// TIA Portal V19 export
FUNCTION_BLOCK "A0302_Manipolatore_FB"   // FB78, LAD
// stored: MemoryReserve 100, SetENOAutomatically false
   VAR_INPUT
      AreaInterface : "AreaInterface";
      ZSI : "udt_ZoneSafetyInterface";
      DSI_Testa_Feed : "udt_DeviceSafetyInterface";
      DSI_Coda_Feed : "udt_DeviceSafetyInterface";
      DSI_Valve : "udt_DeviceSafetyInterface";
      Drive_Testa : "TAx_DriveInterface";
      Drive_Coda : "TAx_DriveInterface";
      DataIn : Struct
         OP_MoveToPos : Bool;
         Sollevamento : Struct
            OP : "OP_PB";
         END_STRUCT;
         Magneti : Struct
            OP : "OP_PB";
         END_STRUCT;
         Sens : Struct
            Ls1 : Bool;   // Banco di controllo - Ls 1 controllo accumulo pezzi scivolo 1
            Ls2 : Bool;   // Banco di controllo - Ls 2 controllo accumulo pezzi scivolo 2
            Ls3 : Bool;   // Banco di controllo - Ls 3 controllo accumulo pezzi scivolo 3
            Ls4 : Bool;   // Banco di controllo - Ls 4 controllo accumulo pezzi scivolo 4
         END_STRUCT;
      END_STRUCT;
      CIn : Struct
         Manager : Struct
            EnableStopDoorOpeningReq { ExternalAccessible := 'False'; ExternalVisible := 'False'; ExternalWritable := 'False'} : Bool;
            EnableStopInPhase { ExternalAccessible := 'False'; ExternalVisible := 'False'; ExternalWritable := 'False'} : Bool;
            EnableStopProgrammed { ExternalAccessible := 'False'; ExternalVisible := 'False'; ExternalWritable := 'False'} : Bool;
            Control_ON { ExternalAccessible := 'False'; ExternalVisible := 'False'; ExternalWritable := 'False'} : Bool;
            MoveToPos { ExternalAccessible := 'False'; ExternalVisible := 'False'; ExternalWritable := 'False'} : Bool;
            Pos { ExternalAccessible := 'False'; ExternalVisible := 'False'; ExternalWritable := 'False'} : LReal;
            Vel : LReal;
            Acc : LReal;
            Dec : LReal;
            Sollevamento { ExternalAccessible := 'False'; ExternalVisible := 'False'; ExternalWritable := 'False'} : Struct
               Rest : Bool;
               Work : Bool;
            END_STRUCT;
            Magneti { ExternalAccessible := 'False'; ExternalVisible := 'False'; ExternalWritable := 'False'} : Struct
               Rest : Bool;
               Work : Bool;
            END_STRUCT;
         END_STRUCT;
         OP_SemiAut_PB { ExternalWritable := 'False'} : Bool;
         Rulliera { ExternalWritable := 'False'} : Struct
            Centratori : "ValveMachine_COut";
            Coda : Struct
               Sens : Struct
                  FTC_Rall : Bool;   // Sensori presenza materiale banco rallentamento ingresso
                  FTC_Prox_Ing : Bool;   // Sensori presenza materiale banco limite ingresso
               END_STRUCT;
            END_STRUCT;
            Centro : Struct
               Sens : Struct
                  FTC_Centrale : Bool;   // 2010BF1 - I50.2
               END_STRUCT;
            END_STRUCT;
         END_STRUCT;
         CarroPareggTesta { ExternalWritable := 'False'} : Struct
            Sens : Struct
               FTC1_Rall : Bool;   // 2010BF2 - I50.3
               FTC2_Prox_Ls : Bool;   // 2010BF3 - I50.4
               PresenzaMat : Bool;   // FC presenza materiale agganciato lato paregg testa
            END_STRUCT;
         END_STRUCT;
         CarroPareggCoda { ExternalWritable := 'False'} : Struct
            Sens : Struct
               FTC_Ingombro_In : Bool;   // 2012BF1 - I50.0
               FTC_Ingombro_Out : Bool;   // 2012BF2 - I50.1
               PresenzaMat : Bool;   // FC presenza materiale agganciato lato paregg coda
            END_STRUCT;
         END_STRUCT;
         CarriPareggiatori : Struct
            ZoneA0302Entry_Empty { ExternalWritable := 'False'} : Bool;
            ZoneA0302Exit_Empty { ExternalWritable := 'False'} : Bool;
            RequestNewPosition : Bool;
         END_STRUCT;
         Spalle : Struct
            Coda : Struct
               ActualPos : LReal;
            END_STRUCT;
            Testa : Struct
               ActualPos : LReal;
            END_STRUCT;
         END_STRUCT;
      END_STRUCT;
      Config : Struct
         Testa : Struct
            Ax : "Positioning_EPOS_Machine_Config_NEW";
            Sollevatore : "ValveMachine_Config";
            Magnete : "ValveMachine_Config";
         END_STRUCT;
         Coda : Struct
            Ax : "Positioning_EPOS_Machine_Config_NEW";
            Sollevatore : "ValveMachine_Config";
            Magnete : "ValveMachine_Config";
         END_STRUCT;
         DelayMissingCondition : Time;
      END_STRUCT;
      HWID_AxTesta_TEL111 : HW_SUBMODULE;
      HWID_AxCoda_TEL111 : HW_SUBMODULE;
   END_VAR
   VAR_OUTPUT
      MachineInterface : "MachineInterface";
      COut : Struct
         Testa : Struct
            Ax : "Positioning_EPOS_Machine_COut";
            Sollevatore : "ValveMachine_COut";
            Magnete : "ValveMachine_COut";
         END_STRUCT;
         Coda : Struct
            Ax : "Positioning_EPOS_Machine_COut";
            Sollevatore : "ValveMachine_COut";
            Magnete : "ValveMachine_COut";
         END_STRUCT;
         CheckAxTesta : Struct
            InPos_Prelievo : Bool;
            InPos_BancoScarto : Bool;
            InPos_BancoA0303 : Bool;
         END_STRUCT;
         CheckAxCoda : Struct
            InPos_Prelievo : Bool;
            InPos_BancoScarto : Bool;
            InPos_BancoA0303 : Bool;
         END_STRUCT;
         InPos_Prelievo : Bool;
         InPos_BancoScarto : Bool;
         InPos_BancoA0303 : Bool;
         OutWorkSpace : Bool;   // Fuori ingombro banco A0303
      END_STRUCT;
   END_VAR
   VAR_IN_OUT
      Par : Struct
         Ax : "Positioning_EPOS_Machine_Par";
         Ax_Aut : "A0301_Mach_Speed_Par";
         Ax_Pos : Struct
            Prelievo : LReal;
            BancoCtrl : LReal;
            BancoA0303 : LReal;
            Tollerance : Struct
               Prelievo : LReal;
               BancoCtrl : LReal;
               BancoA0303 : LReal;
            END_STRUCT;
         END_STRUCT;
      END_STRUCT;
      Pers_Data : Struct
         EncoderAbsolute_Preset_OK : Bool;
         Persistent_ActualPosition : LReal;
      END_STRUCT;
   END_VAR
   VAR
      Alarm : Struct
         Testa : Struct
            Ax : "Positioning_EPOS_Machine_Alr";
            Sollevatore : "ValveAlr";
            Magnete : "ValveAlr";
         END_STRUCT;
         Coda : Struct
            Ax : "Positioning_EPOS_Machine_Alr";
            Sollevatore : "ValveAlr";
            Magnete : "ValveAlr";
         END_STRUCT;
         CheckBothAxMove : Bool;
      END_STRUCT;
      Warning : Struct
         Testa : Struct
            Ax : "Positioning_EPOS_Machine_Wng";
            Sollevatore : "ValveMachine_Wng";
            Magnete : "ValveMachine_Wng";
         END_STRUCT;
         Coda : Struct
            Ax : "Positioning_EPOS_Machine_Wng";
            Sollevatore : "ValveMachine_Wng";
            Magnete : "ValveMachine_Wng";
         END_STRUCT;
         MissingCnd : Struct
            OP_REST_Sollevamento : Bool;   // Mancanza comando arresto
            OP_WORK_Sollevamento : Bool;   // Mancanza consenso lavoro
            OP_REST_Magneti : Bool;   // Mancanza comando arresto
            OP_WORK_Magneti : Bool;   // Mancanza consenso lavoro
         END_STRUCT;
      END_STRUCT;
      HMI : Struct
         Selection : Struct   // 0=Disable / 1=Enable Pin
            Ax : Int;   // 0:Entrambe / 1:Testa / 2:Coda
         END_STRUCT;
         Ax_Testa : "AnalogSens_HmiData";
         Ax_Coda : "AnalogSens_HmiData";
      END_STRUCT;
      Sts : Struct
         ReadyForMove : Bool;   // Pronto al movimento
         OP_Manip_CanMoveFreely : Bool;
         OP_Ax_CanMoveFreely : Bool;
         Op_MoveToPos_Cnd : Bool;
         Sollevamento : Struct
            OP_Rest_Cnd : Bool;
            Op_Work_Cnd : Bool;
         END_STRUCT;
         Magneti : Struct
            OP_Rest_Cnd : Bool;
            Op_Work_Cnd : Bool;
         END_STRUCT;
         Coda_PermessoDaSynchOk : Bool;
         Testa_PermessoDaSynchOk : Bool;
      END_STRUCT;
      Ctrl : Struct
         Sollevamento : Struct
            OP_Rest_Man : Bool;
            OP_Work_Man : Bool;
            OP_Rest_Aut : Bool;
            OP_Work_Aut : Bool;
            OP_Rest : Bool;
            OP_Work : Bool;
         END_STRUCT;
         Magneti : Struct
            OP_Rest_Aut : Bool;
            OP_Work_Aut : Bool;
            OP_Rest_Man : Bool;
            OP_Work_Man : Bool;
            OP_Rest : Bool;
            OP_Work : Bool;
         END_STRUCT;
         Ax : Struct
            OP_MoveToPos_Man : Bool;
            OP_MoveToPos_Aut : Bool;
            OP_MoveToPos : Bool;
         END_STRUCT;
      END_STRUCT;
      AUX : Struct
         OP_MoveToPos : Bool;
         Sollevamento : Struct
            OP_Rest : Bool;
            OP_Work : Bool;
         END_STRUCT;
         Magneti : Struct
            OP_Rest : Bool;
            OP_Work : Bool;
         END_STRUCT;
      END_STRUCT;
      Ax_Testa : "Positioning_EPOS_Machine_FB_NEW";
      Ax_Coda : "Positioning_EPOS_Machine_FB_NEW";
      Sollevatore_Testa { S7_SetPoint := 'True'} : "ValveMachine_FB";
      Sollevatore_Coda { S7_SetPoint := 'True'} : "ValveMachine_FB";
      Magnete_Testa { S7_SetPoint := 'True'} : "ValveMachine_FB";
      Magnete_Coda { S7_SetPoint := 'True'} : "ValveMachine_FB";
      TON_Magneti : Struct
         OP_REST_MissingCnd { S7_SetPoint := 'True'} : TON_TIME;
         OP_WORK_MissingCnd { S7_SetPoint := 'True'} : TON_TIME;
      END_STRUCT;
      TON_Sollevamento : Struct
         OP_REST_MissingCnd { S7_SetPoint := 'True'} : TON_TIME;
         OP_WORK_MissingCnd { S7_SetPoint := 'True'} : TON_TIME;
      END_STRUCT;
      TON_CheckAxMove : IEC_TIMER;
      CheckAxisSynch { ExternalAccessible := 'False'; ExternalVisible := 'False'; ExternalWritable := 'False'} : "CheckAxisSynch";
      Sts_PosAxis { S7_SetPoint := 'True'} : Int;
   END_VAR
   VAR_TEMP
      PE : Struct
         OP_MoveToPos : Bool;
         Sollevamento : Struct
            OP_Rest : Bool;
            OP_Work : Bool;
         END_STRUCT;
         Magneti : Struct
            OP_Rest : Bool;
            OP_Work : Bool;
         END_STRUCT;
      END_STRUCT;
   END_VAR
   VAR CONSTANT
      MaxDistance : LReal := 5.0;
      MinDistance : LReal := 0.7;   // soglia inferiore per isteresi
   END_VAR
   VAR_TEMP   // added for the SCL form of the ladder/FBD networks
      _w1 : Bool;
      _w2 : Bool;
      _w3 : Bool;
      _w4 : Bool;
      _w5 : Bool;
      _w6 : Bool;
      _w7 : Bool;
      _w8 : Bool;
      _w9 : Bool;
   END_VAR
BEGIN

REGION Network 1 (SCL): Reset allarmi
   IF #AreaInterface.RstAlarms THEN
       #Alarm.CheckBothAxMove:=FALSE;
       #Warning.Testa.Ax.Minus_CndMissing := FALSE;
       #Warning.Testa.Ax.Plus_CndMissing := FALSE;
       #Warning.Coda.Ax.Minus_CndMissing := FALSE;
       #Warning.Coda.Ax.Plus_CndMissing := FALSE;
   END_IF;
END_REGION

REGION Network 3 (SCL): PrjConfig - GESTIONE PARAMETRI MANIPOLATORI
   // Asse MANIPOLATORI









   // SOLLEVATORE
   // 







   // MAGNETE
   //
END_REGION

REGION Network 5: [Ax] - Controllo posizione dei Manipolatori In PRELIEVO su PAREGGIATORI
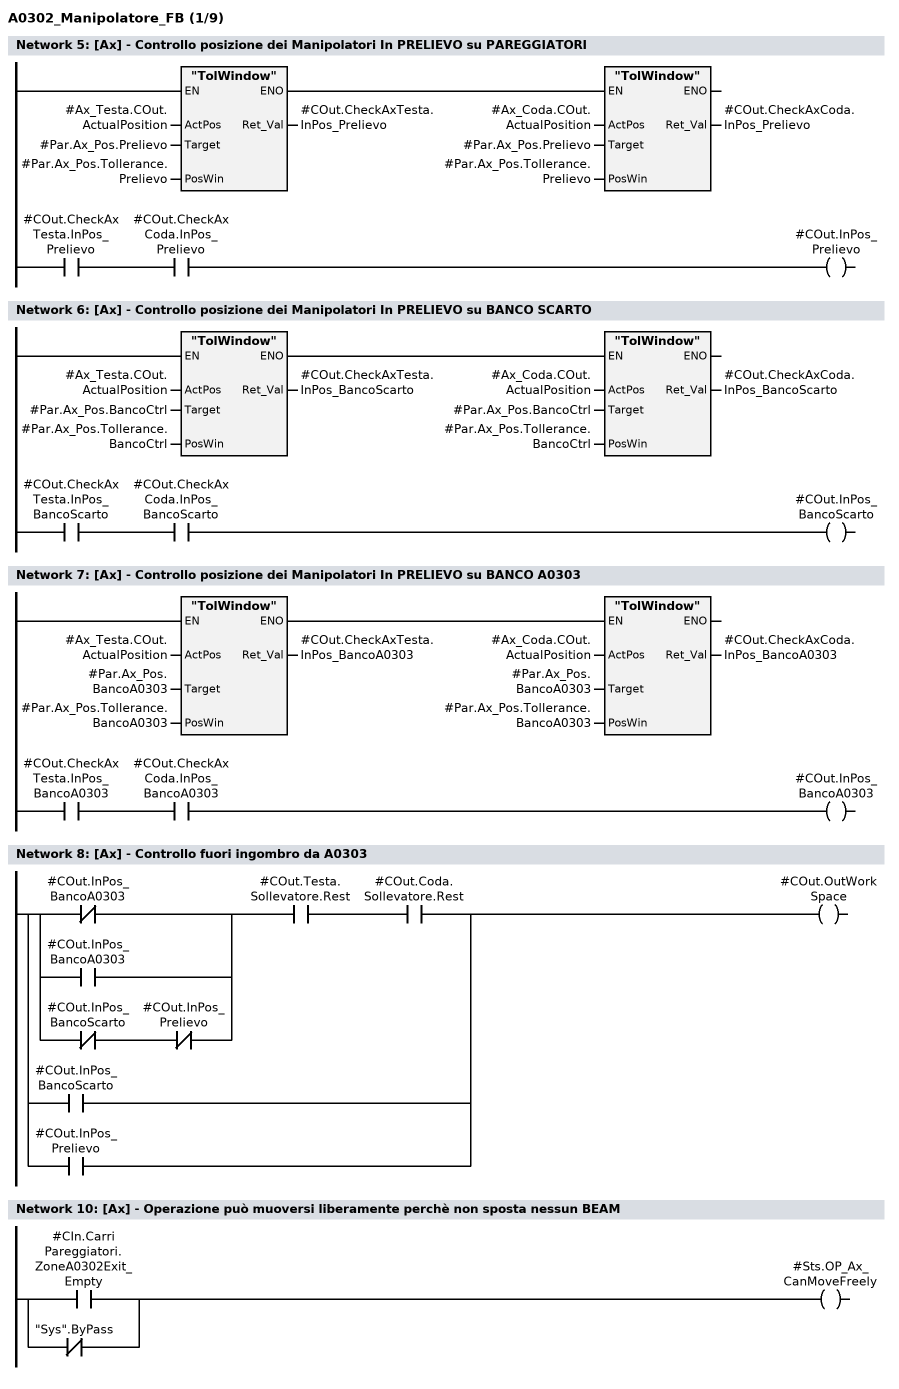
   RUNG wire#powerrail
      "TolWindow"(ActPos := #Ax_Testa.COut.ActualPosition, Target := #Par.Ax_Pos.Prelievo, PosWin := #Par.Ax_Pos.Tollerance.Prelievo, Ret_Val => #COut.CheckAxTesta.InPos_Prelievo)
      "TolWindow"(ActPos := #Ax_Coda.COut.ActualPosition, Target := #Par.Ax_Pos.Prelievo, PosWin := #Par.Ax_Pos.Tollerance.Prelievo, Ret_Val => #COut.CheckAxCoda.InPos_Prelievo)
   END_RUNG
   RUNG wire#powerrail
      Contact( #COut.CheckAxTesta.InPos_Prelievo )
      Contact( #COut.CheckAxCoda.InPos_Prelievo )
      Coil( #COut.InPos_Prelievo )
   END_RUNG
   // the same network as SCL:
   #COut.CheckAxTesta.InPos_Prelievo := "TolWindow"(ActPos := #Ax_Testa.COut.ActualPosition,
                           Target := #Par.Ax_Pos.Prelievo,
                           PosWin := #Par.Ax_Pos.Tollerance.Prelievo,
                           ENO => #_w1);
   IF #_w1 THEN
       #COut.CheckAxCoda.InPos_Prelievo := "TolWindow"(ActPos := #Ax_Coda.COut.ActualPosition,
                               Target := #Par.Ax_Pos.Prelievo,
                               PosWin := #Par.Ax_Pos.Tollerance.Prelievo);
   END_IF;
   #COut.InPos_Prelievo := #COut.CheckAxTesta.InPos_Prelievo AND #COut.CheckAxCoda.InPos_Prelievo;
END_REGION

REGION Network 6: [Ax] - Controllo posizione dei Manipolatori In PRELIEVO su BANCO SCARTO
   RUNG wire#powerrail
      "TolWindow"(ActPos := #Ax_Testa.COut.ActualPosition, Target := #Par.Ax_Pos.BancoCtrl, PosWin := #Par.Ax_Pos.Tollerance.BancoCtrl, Ret_Val => #COut.CheckAxTesta.InPos_BancoScarto)
      "TolWindow"(ActPos := #Ax_Coda.COut.ActualPosition, Target := #Par.Ax_Pos.BancoCtrl, PosWin := #Par.Ax_Pos.Tollerance.BancoCtrl, Ret_Val => #COut.CheckAxCoda.InPos_BancoScarto)
   END_RUNG
   RUNG wire#powerrail
      Contact( #COut.CheckAxTesta.InPos_BancoScarto )
      Contact( #COut.CheckAxCoda.InPos_BancoScarto )
      Coil( #COut.InPos_BancoScarto )
   END_RUNG
   // the same network as SCL:
   #COut.CheckAxTesta.InPos_BancoScarto := "TolWindow"(ActPos := #Ax_Testa.COut.ActualPosition,
                           Target := #Par.Ax_Pos.BancoCtrl,
                           PosWin := #Par.Ax_Pos.Tollerance.BancoCtrl,
                           ENO => #_w1);
   IF #_w1 THEN
       #COut.CheckAxCoda.InPos_BancoScarto := "TolWindow"(ActPos := #Ax_Coda.COut.ActualPosition,
                               Target := #Par.Ax_Pos.BancoCtrl,
                               PosWin := #Par.Ax_Pos.Tollerance.BancoCtrl);
   END_IF;
   #COut.InPos_BancoScarto := #COut.CheckAxTesta.InPos_BancoScarto AND #COut.CheckAxCoda.InPos_BancoScarto;
END_REGION

REGION Network 7: [Ax] - Controllo posizione dei Manipolatori In PRELIEVO su BANCO A0303
   RUNG wire#powerrail
      "TolWindow"(ActPos := #Ax_Testa.COut.ActualPosition, Target := #Par.Ax_Pos.BancoA0303, PosWin := #Par.Ax_Pos.Tollerance.BancoA0303, Ret_Val => #COut.CheckAxTesta.InPos_BancoA0303)
      "TolWindow"(ActPos := #Ax_Coda.COut.ActualPosition, Target := #Par.Ax_Pos.BancoA0303, PosWin := #Par.Ax_Pos.Tollerance.BancoA0303, Ret_Val => #COut.CheckAxCoda.InPos_BancoA0303)
   END_RUNG
   RUNG wire#powerrail
      Contact( #COut.CheckAxTesta.InPos_BancoA0303 )
      Contact( #COut.CheckAxCoda.InPos_BancoA0303 )
      Coil( #COut.InPos_BancoA0303 )
   END_RUNG
   // the same network as SCL:
   #COut.CheckAxTesta.InPos_BancoA0303 := "TolWindow"(ActPos := #Ax_Testa.COut.ActualPosition,
                           Target := #Par.Ax_Pos.BancoA0303,
                           PosWin := #Par.Ax_Pos.Tollerance.BancoA0303,
                           ENO => #_w1);
   IF #_w1 THEN
       #COut.CheckAxCoda.InPos_BancoA0303 := "TolWindow"(ActPos := #Ax_Coda.COut.ActualPosition,
                               Target := #Par.Ax_Pos.BancoA0303,
                               PosWin := #Par.Ax_Pos.Tollerance.BancoA0303);
   END_IF;
   #COut.InPos_BancoA0303 := #COut.CheckAxTesta.InPos_BancoA0303 AND #COut.CheckAxCoda.InPos_BancoA0303;
END_REGION

REGION Network 8: [Ax] - Controllo fuori ingombro da A0303
   RUNG wire#powerrail
      I_Contact( #COut.InPos_BancoA0303 )
      wire#w1
      Contact( #COut.Testa.Sollevatore.Rest )
      Contact( #COut.Coda.Sollevatore.Rest )
      wire#w2
      Coil( #COut.OutWorkSpace )
   END_RUNG
   RUNG wire#powerrail
      Contact( #COut.InPos_BancoA0303 )
   END_RUNG wire#w1
   RUNG wire#powerrail
      I_Contact( #COut.InPos_BancoScarto )
      I_Contact( #COut.InPos_Prelievo )
   END_RUNG wire#w1
   RUNG wire#powerrail
      Contact( #COut.InPos_BancoScarto )
   END_RUNG wire#w2
   RUNG wire#powerrail
      Contact( #COut.InPos_Prelievo )
   END_RUNG wire#w2
   // the same network as SCL:
   #COut.OutWorkSpace := ((NOT #COut.InPos_BancoA0303 OR #COut.InPos_BancoA0303 OR (NOT #COut.InPos_BancoScarto AND NOT #COut.InPos_Prelievo)) AND #COut.Testa.Sollevatore.Rest AND #COut.Coda.Sollevatore.Rest) OR #COut.InPos_BancoScarto OR #COut.InPos_Prelievo;
END_REGION

REGION Network 10: [Ax] - Operazione può muoversi liberamente perchè non sposta nessun BEAM
   RUNG wire#powerrail
      Contact( #CIn.CarriPareggiatori.ZoneA0302Exit_Empty )
      wire#w1
      Coil( #Sts.OP_Ax_CanMoveFreely )
   END_RUNG
   RUNG wire#powerrail
      I_Contact( "Sys".ByPass )
   END_RUNG wire#w1
   // the same network as SCL:
   #Sts.OP_Ax_CanMoveFreely := #CIn.CarriPareggiatori.ZoneA0302Exit_Empty OR NOT "Sys".ByPass;
END_REGION

REGION Network 11: [Ax] - Comando Operazione Lavoro / Riposo (AUT)
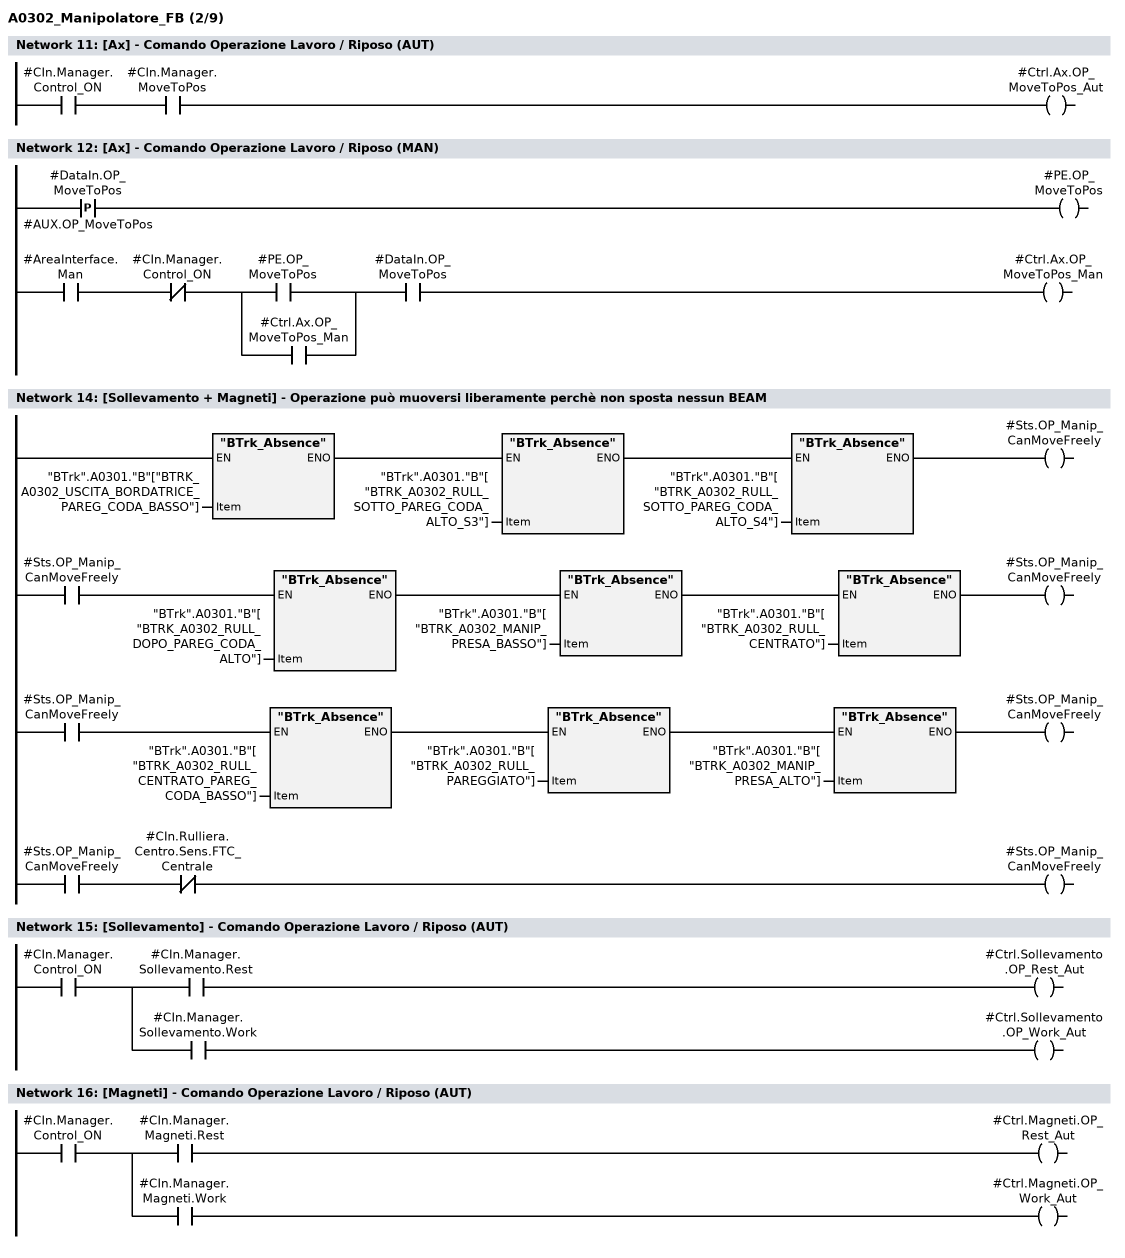
   RUNG wire#powerrail
      Contact( #CIn.Manager.Control_ON )
      Contact( #CIn.Manager.MoveToPos )
      Coil( #Ctrl.Ax.OP_MoveToPos_Aut )
   END_RUNG
   // the same network as SCL:
   #Ctrl.Ax.OP_MoveToPos_Aut := #CIn.Manager.Control_ON AND #CIn.Manager.MoveToPos;
END_REGION

REGION Network 12: [Ax] - Comando Operazione Lavoro / Riposo (MAN)
   RUNG wire#powerrail
      P_Contact(operand := #DataIn.OP_MoveToPos, bit := #AUX.OP_MoveToPos)
      Coil( #PE.OP_MoveToPos )
   END_RUNG
   RUNG wire#powerrail
      Contact( #AreaInterface.Man )
      I_Contact( #CIn.Manager.Control_ON )
      wire#w1
      Contact( #PE.OP_MoveToPos )
      wire#w2
      Contact( #DataIn.OP_MoveToPos )
      Coil( #Ctrl.Ax.OP_MoveToPos_Man )
   END_RUNG
   RUNG wire#w1
      Contact( #Ctrl.Ax.OP_MoveToPos_Man )
   END_RUNG wire#w2
   // the same network as SCL:
   #_w1 := #DataIn.OP_MoveToPos AND NOT #AUX.OP_MoveToPos;   // rising edge of #DataIn.OP_MoveToPos
   #AUX.OP_MoveToPos := #DataIn.OP_MoveToPos;
   #PE.OP_MoveToPos := #_w1;
   #Ctrl.Ax.OP_MoveToPos_Man := #AreaInterface.Man AND NOT #CIn.Manager.Control_ON AND (#PE.OP_MoveToPos OR #Ctrl.Ax.OP_MoveToPos_Man) AND #DataIn.OP_MoveToPos;
END_REGION

REGION Network 13: <+>
END_REGION

REGION Network 14: [Sollevamento + Magneti] - Operazione può muoversi liberamente perchè non sposta nessun BEAM
   RUNG wire#powerrail
      "BTrk_Absence"(Item := "BTrk".A0301."B"["BTRK_A0302_USCITA_BORDATRICE_PAREG_CODA_BASSO"])
      "BTrk_Absence"(Item := "BTrk".A0301."B"["BTRK_A0302_RULL_SOTTO_PAREG_CODA_ALTO_S3"])
      "BTrk_Absence"(Item := "BTrk".A0301."B"["BTRK_A0302_RULL_SOTTO_PAREG_CODA_ALTO_S4"])
      Coil( #Sts.OP_Manip_CanMoveFreely )
   END_RUNG
   RUNG wire#powerrail
      Contact( #Sts.OP_Manip_CanMoveFreely )
      "BTrk_Absence"(Item := "BTrk".A0301."B"["BTRK_A0302_RULL_DOPO_PAREG_CODA_ALTO"])
      "BTrk_Absence"(Item := "BTrk".A0301."B"["BTRK_A0302_MANIP_PRESA_BASSO"])
      "BTrk_Absence"(Item := "BTrk".A0301."B"["BTRK_A0302_RULL_CENTRATO"])
      Coil( #Sts.OP_Manip_CanMoveFreely )
   END_RUNG
   RUNG wire#powerrail
      Contact( #Sts.OP_Manip_CanMoveFreely )
      "BTrk_Absence"(Item := "BTrk".A0301."B"["BTRK_A0302_RULL_CENTRATO_PAREG_CODA_BASSO"])
      "BTrk_Absence"(Item := "BTrk".A0301."B"["BTRK_A0302_RULL_PAREGGIATO"])
      "BTrk_Absence"(Item := "BTrk".A0301."B"["BTRK_A0302_MANIP_PRESA_ALTO"])
      Coil( #Sts.OP_Manip_CanMoveFreely )
   END_RUNG
   RUNG wire#powerrail
      Contact( #Sts.OP_Manip_CanMoveFreely )
      I_Contact( #CIn.Rulliera.Centro.Sens.FTC_Centrale )
      Coil( #Sts.OP_Manip_CanMoveFreely )
   END_RUNG
   // the same network as SCL:
   "BTrk_Absence"(Item := "BTrk".A0301."B"["BTRK_A0302_USCITA_BORDATRICE_PAREG_CODA_BASSO"], ENO => #_w1);
   "BTrk_Absence"(EN := #_w1, Item := "BTrk".A0301."B"["BTRK_A0302_RULL_SOTTO_PAREG_CODA_ALTO_S3"], ENO => #_w2);
   "BTrk_Absence"(EN := #_w2, Item := "BTrk".A0301."B"["BTRK_A0302_RULL_SOTTO_PAREG_CODA_ALTO_S4"], ENO => #_w3);
   #Sts.OP_Manip_CanMoveFreely := #_w3;
   "BTrk_Absence"(EN := #Sts.OP_Manip_CanMoveFreely,
                  Item := "BTrk".A0301."B"["BTRK_A0302_RULL_DOPO_PAREG_CODA_ALTO"],
                  ENO => #_w4);
   "BTrk_Absence"(EN := #_w4, Item := "BTrk".A0301."B"["BTRK_A0302_MANIP_PRESA_BASSO"], ENO => #_w5);
   "BTrk_Absence"(EN := #_w5, Item := "BTrk".A0301."B"["BTRK_A0302_RULL_CENTRATO"], ENO => #_w6);
   #Sts.OP_Manip_CanMoveFreely := #_w6;
   "BTrk_Absence"(EN := #Sts.OP_Manip_CanMoveFreely,
                  Item := "BTrk".A0301."B"["BTRK_A0302_RULL_CENTRATO_PAREG_CODA_BASSO"],
                  ENO => #_w7);
   "BTrk_Absence"(EN := #_w7, Item := "BTrk".A0301."B"["BTRK_A0302_RULL_PAREGGIATO"], ENO => #_w8);
   "BTrk_Absence"(EN := #_w8, Item := "BTrk".A0301."B"["BTRK_A0302_MANIP_PRESA_ALTO"], ENO => #_w9);
   #Sts.OP_Manip_CanMoveFreely := #_w9;
   #Sts.OP_Manip_CanMoveFreely := #Sts.OP_Manip_CanMoveFreely AND NOT #CIn.Rulliera.Centro.Sens.FTC_Centrale;
END_REGION

REGION Network 15: [Sollevamento] - Comando Operazione Lavoro / Riposo (AUT)
   RUNG wire#powerrail
      Contact( #CIn.Manager.Control_ON )
      wire#w1
      Contact( #CIn.Manager.Sollevamento.Rest )
      Coil( #Ctrl.Sollevamento.OP_Rest_Aut )
   END_RUNG
   RUNG wire#w1
      Contact( #CIn.Manager.Sollevamento.Work )
      Coil( #Ctrl.Sollevamento.OP_Work_Aut )
   END_RUNG
   // the same network as SCL:
   #Ctrl.Sollevamento.OP_Rest_Aut := #CIn.Manager.Control_ON AND #CIn.Manager.Sollevamento.Rest;
   #Ctrl.Sollevamento.OP_Work_Aut := #CIn.Manager.Control_ON AND #CIn.Manager.Sollevamento.Work;
END_REGION

REGION Network 16: [Magneti] - Comando Operazione Lavoro / Riposo (AUT)
   RUNG wire#powerrail
      Contact( #CIn.Manager.Control_ON )
      wire#w1
      Contact( #CIn.Manager.Magneti.Rest )
      Coil( #Ctrl.Magneti.OP_Rest_Aut )
   END_RUNG
   RUNG wire#w1
      Contact( #CIn.Manager.Magneti.Work )
      Coil( #Ctrl.Magneti.OP_Work_Aut )
   END_RUNG
   // the same network as SCL:
   #Ctrl.Magneti.OP_Rest_Aut := #CIn.Manager.Control_ON AND #CIn.Manager.Magneti.Rest;
   #Ctrl.Magneti.OP_Work_Aut := #CIn.Manager.Control_ON AND #CIn.Manager.Magneti.Work;
END_REGION

REGION Network 17: <+>
END_REGION

REGION Network 18: [Sollevamento] - Comando Operazione Lavoro / Riposo (MAN)
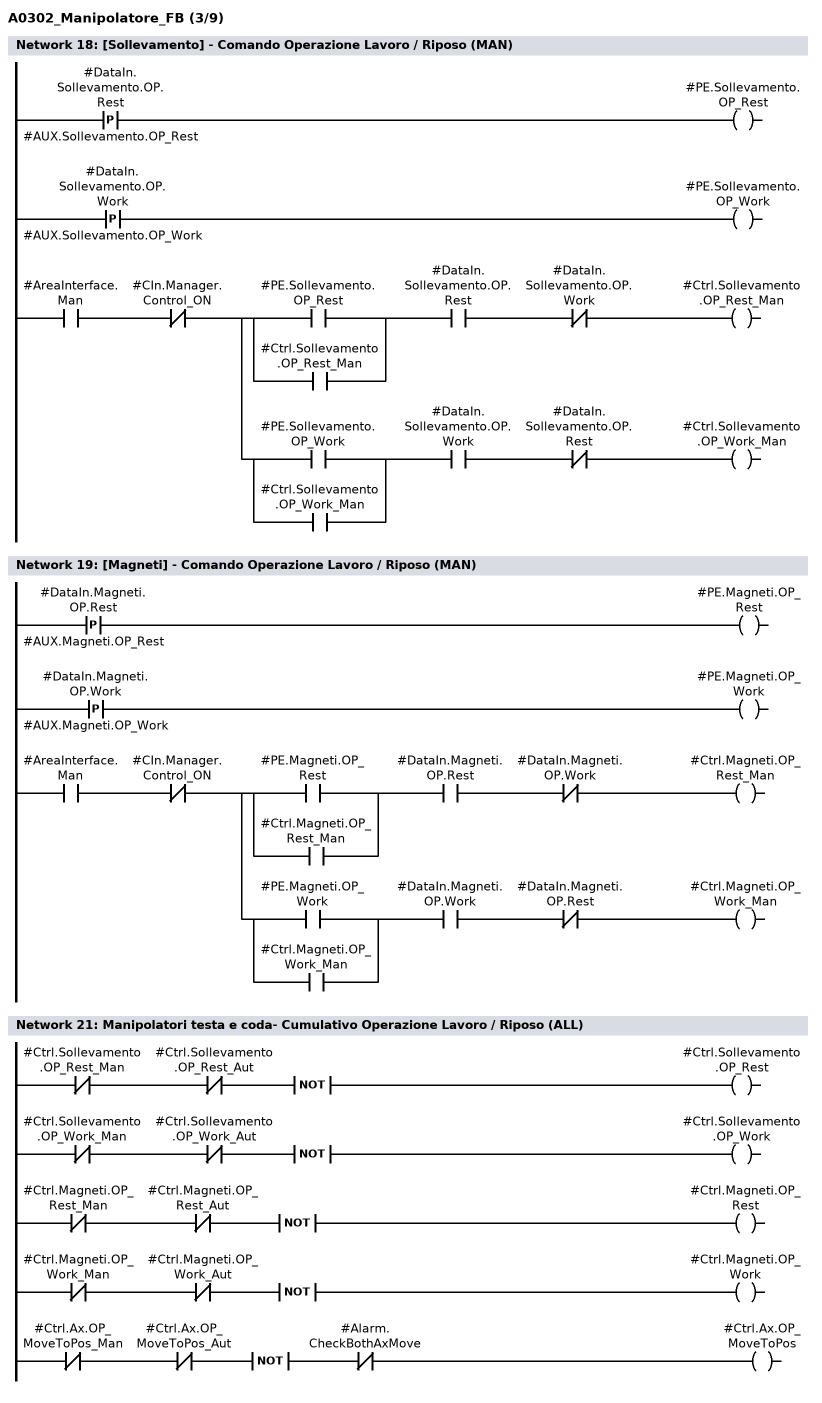
   RUNG wire#powerrail
      P_Contact(operand := #DataIn.Sollevamento.OP.Rest, bit := #AUX.Sollevamento.OP_Rest)
      Coil( #PE.Sollevamento.OP_Rest )
   END_RUNG
   RUNG wire#powerrail
      P_Contact(operand := #DataIn.Sollevamento.OP.Work, bit := #AUX.Sollevamento.OP_Work)
      Coil( #PE.Sollevamento.OP_Work )
   END_RUNG
   RUNG wire#powerrail
      Contact( #AreaInterface.Man )
      I_Contact( #CIn.Manager.Control_ON )
      wire#w1
      Contact( #PE.Sollevamento.OP_Rest )
      wire#w2
      Contact( #DataIn.Sollevamento.OP.Rest )
      I_Contact( #DataIn.Sollevamento.OP.Work )
      Coil( #Ctrl.Sollevamento.OP_Rest_Man )
   END_RUNG
   RUNG wire#w1
      Contact( #Ctrl.Sollevamento.OP_Rest_Man )
   END_RUNG wire#w2
   RUNG wire#w1
      Contact( #PE.Sollevamento.OP_Work )
      wire#w3
      Contact( #DataIn.Sollevamento.OP.Work )
      I_Contact( #DataIn.Sollevamento.OP.Rest )
      Coil( #Ctrl.Sollevamento.OP_Work_Man )
   END_RUNG
   RUNG wire#w1
      Contact( #Ctrl.Sollevamento.OP_Work_Man )
   END_RUNG wire#w3
   // the same network as SCL:
   #_w1 := #DataIn.Sollevamento.OP.Rest AND NOT #AUX.Sollevamento.OP_Rest;   // rising edge of #DataIn.Sollevamento.OP.Rest
   #AUX.Sollevamento.OP_Rest := #DataIn.Sollevamento.OP.Rest;
   #PE.Sollevamento.OP_Rest := #_w1;
   #_w2 := #DataIn.Sollevamento.OP.Work AND NOT #AUX.Sollevamento.OP_Work;   // rising edge of #DataIn.Sollevamento.OP.Work
   #AUX.Sollevamento.OP_Work := #DataIn.Sollevamento.OP.Work;
   #PE.Sollevamento.OP_Work := #_w2;
   #_w3 := #AreaInterface.Man AND NOT #CIn.Manager.Control_ON;
   #Ctrl.Sollevamento.OP_Rest_Man := #_w3 AND (#PE.Sollevamento.OP_Rest OR #Ctrl.Sollevamento.OP_Rest_Man) AND #DataIn.Sollevamento.OP.Rest AND NOT #DataIn.Sollevamento.OP.Work;
   #Ctrl.Sollevamento.OP_Work_Man := #_w3 AND (#PE.Sollevamento.OP_Work OR #Ctrl.Sollevamento.OP_Work_Man) AND #DataIn.Sollevamento.OP.Work AND NOT #DataIn.Sollevamento.OP.Rest;
END_REGION

REGION Network 19: [Magneti] - Comando Operazione Lavoro / Riposo (MAN)
   RUNG wire#powerrail
      P_Contact(operand := #DataIn.Magneti.OP.Rest, bit := #AUX.Magneti.OP_Rest)
      Coil( #PE.Magneti.OP_Rest )
   END_RUNG
   RUNG wire#powerrail
      P_Contact(operand := #DataIn.Magneti.OP.Work, bit := #AUX.Magneti.OP_Work)
      Coil( #PE.Magneti.OP_Work )
   END_RUNG
   RUNG wire#powerrail
      Contact( #AreaInterface.Man )
      I_Contact( #CIn.Manager.Control_ON )
      wire#w1
      Contact( #PE.Magneti.OP_Rest )
      wire#w2
      Contact( #DataIn.Magneti.OP.Rest )
      I_Contact( #DataIn.Magneti.OP.Work )
      Coil( #Ctrl.Magneti.OP_Rest_Man )
   END_RUNG
   RUNG wire#w1
      Contact( #Ctrl.Magneti.OP_Rest_Man )
   END_RUNG wire#w2
   RUNG wire#w1
      Contact( #PE.Magneti.OP_Work )
      wire#w3
      Contact( #DataIn.Magneti.OP.Work )
      I_Contact( #DataIn.Magneti.OP.Rest )
      Coil( #Ctrl.Magneti.OP_Work_Man )
   END_RUNG
   RUNG wire#w1
      Contact( #Ctrl.Magneti.OP_Work_Man )
   END_RUNG wire#w3
   // the same network as SCL:
   #_w1 := #DataIn.Magneti.OP.Rest AND NOT #AUX.Magneti.OP_Rest;   // rising edge of #DataIn.Magneti.OP.Rest
   #AUX.Magneti.OP_Rest := #DataIn.Magneti.OP.Rest;
   #PE.Magneti.OP_Rest := #_w1;
   #_w2 := #DataIn.Magneti.OP.Work AND NOT #AUX.Magneti.OP_Work;   // rising edge of #DataIn.Magneti.OP.Work
   #AUX.Magneti.OP_Work := #DataIn.Magneti.OP.Work;
   #PE.Magneti.OP_Work := #_w2;
   #_w3 := #AreaInterface.Man AND NOT #CIn.Manager.Control_ON;
   #Ctrl.Magneti.OP_Rest_Man := #_w3 AND (#PE.Magneti.OP_Rest OR #Ctrl.Magneti.OP_Rest_Man) AND #DataIn.Magneti.OP.Rest AND NOT #DataIn.Magneti.OP.Work;
   #Ctrl.Magneti.OP_Work_Man := #_w3 AND (#PE.Magneti.OP_Work OR #Ctrl.Magneti.OP_Work_Man) AND #DataIn.Magneti.OP.Work AND NOT #DataIn.Magneti.OP.Rest;
END_REGION

REGION Network 20: <+>
END_REGION

REGION Network 21: Manipolatori testa e coda- Cumulativo Operazione Lavoro / Riposo (ALL)
   RUNG wire#powerrail
      I_Contact( #Ctrl.Sollevamento.OP_Rest_Man )
      I_Contact( #Ctrl.Sollevamento.OP_Rest_Aut )
      Not()
      Coil( #Ctrl.Sollevamento.OP_Rest )
   END_RUNG
   RUNG wire#powerrail
      I_Contact( #Ctrl.Sollevamento.OP_Work_Man )
      I_Contact( #Ctrl.Sollevamento.OP_Work_Aut )
      Not()
      Coil( #Ctrl.Sollevamento.OP_Work )
   END_RUNG
   RUNG wire#powerrail
      I_Contact( #Ctrl.Magneti.OP_Rest_Man )
      I_Contact( #Ctrl.Magneti.OP_Rest_Aut )
      Not()
      Coil( #Ctrl.Magneti.OP_Rest )
   END_RUNG
   RUNG wire#powerrail
      I_Contact( #Ctrl.Magneti.OP_Work_Man )
      I_Contact( #Ctrl.Magneti.OP_Work_Aut )
      Not()
      Coil( #Ctrl.Magneti.OP_Work )
   END_RUNG
   RUNG wire#powerrail
      I_Contact( #Ctrl.Ax.OP_MoveToPos_Man )
      I_Contact( #Ctrl.Ax.OP_MoveToPos_Aut )
      Not()
      I_Contact( #Alarm.CheckBothAxMove )
      Coil( #Ctrl.Ax.OP_MoveToPos )
   END_RUNG
   // the same network as SCL:
   #Ctrl.Sollevamento.OP_Rest := NOT (NOT #Ctrl.Sollevamento.OP_Rest_Man AND NOT #Ctrl.Sollevamento.OP_Rest_Aut);
   #Ctrl.Sollevamento.OP_Work := NOT (NOT #Ctrl.Sollevamento.OP_Work_Man AND NOT #Ctrl.Sollevamento.OP_Work_Aut);
   #Ctrl.Magneti.OP_Rest := NOT (NOT #Ctrl.Magneti.OP_Rest_Man AND NOT #Ctrl.Magneti.OP_Rest_Aut);
   #Ctrl.Magneti.OP_Work := NOT (NOT #Ctrl.Magneti.OP_Work_Man AND NOT #Ctrl.Magneti.OP_Work_Aut);
   #Ctrl.Ax.OP_MoveToPos := NOT (NOT #Ctrl.Ax.OP_MoveToPos_Man AND NOT #Ctrl.Ax.OP_MoveToPos_Aut) AND NOT #Alarm.CheckBothAxMove;
END_REGION

REGION Network 22: <+>
END_REGION

REGION Network 23: [Ax] - Condizioni movimento Operazione a Lavoro / Riposo
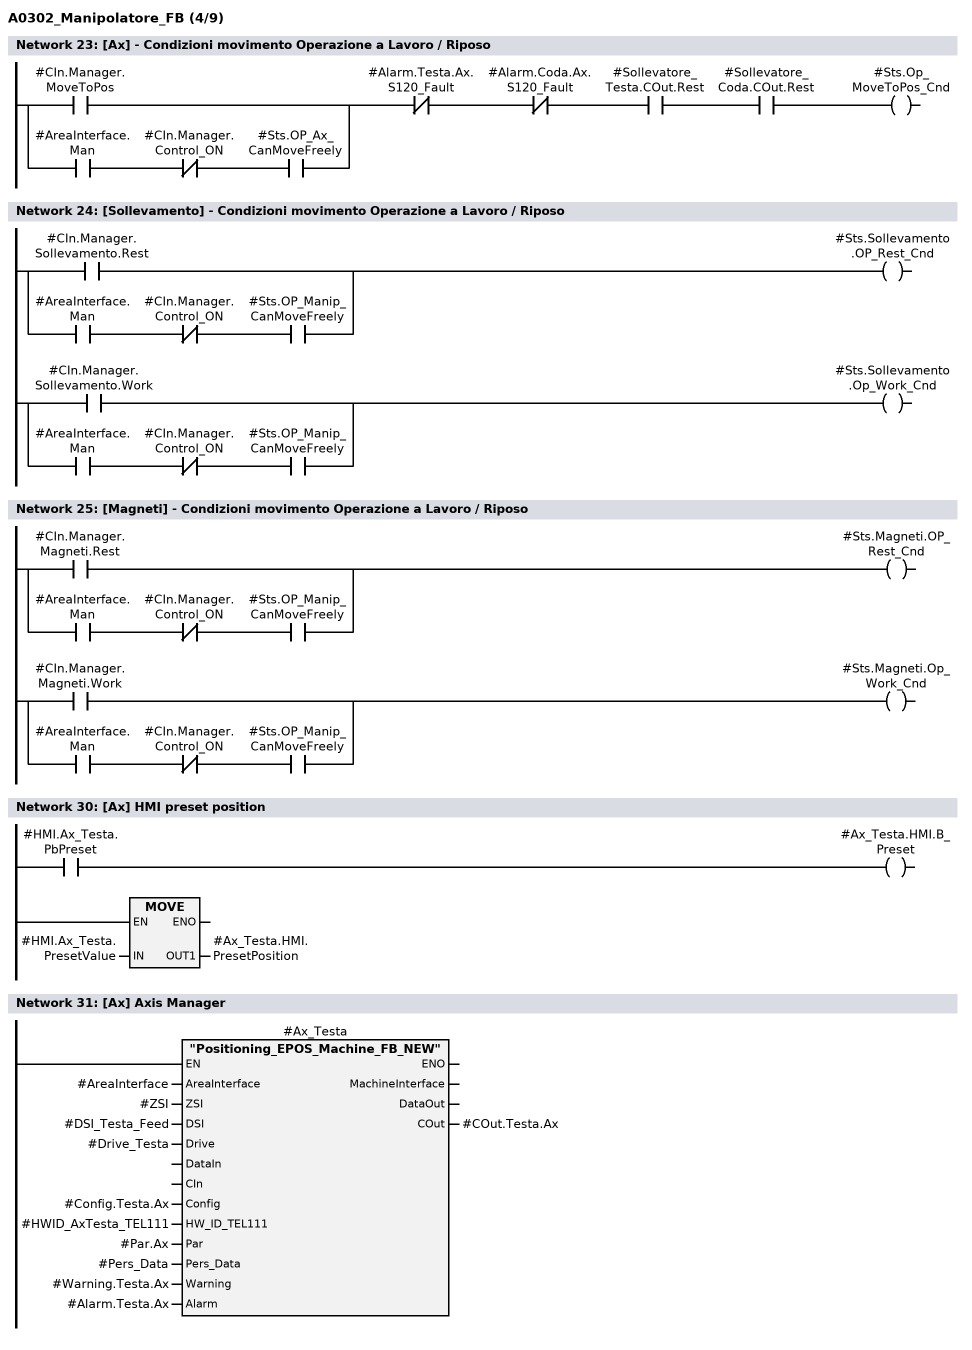
   RUNG wire#powerrail
      Contact( #CIn.Manager.MoveToPos )
      wire#w1
      I_Contact( #Alarm.Testa.Ax.S120_Fault )
      I_Contact( #Alarm.Coda.Ax.S120_Fault )
      Contact( #Sollevatore_Testa.COut.Rest )
      Contact( #Sollevatore_Coda.COut.Rest )
      Coil( #Sts.Op_MoveToPos_Cnd )
   END_RUNG
   RUNG wire#powerrail
      Contact( #AreaInterface.Man )
      I_Contact( #CIn.Manager.Control_ON )
      Contact( #Sts.OP_Ax_CanMoveFreely )
   END_RUNG wire#w1
   // the same network as SCL:
   #Sts.Op_MoveToPos_Cnd := (#CIn.Manager.MoveToPos OR (#AreaInterface.Man AND NOT #CIn.Manager.Control_ON AND #Sts.OP_Ax_CanMoveFreely)) AND NOT #Alarm.Testa.Ax.S120_Fault AND NOT #Alarm.Coda.Ax.S120_Fault AND #Sollevatore_Testa.COut.Rest AND #Sollevatore_Coda.COut.Rest;
END_REGION

REGION Network 24: [Sollevamento] - Condizioni movimento Operazione a Lavoro / Riposo
   RUNG wire#powerrail
      Contact( #CIn.Manager.Sollevamento.Rest )
      wire#w1
      Coil( #Sts.Sollevamento.OP_Rest_Cnd )
   END_RUNG
   RUNG wire#powerrail
      Contact( #AreaInterface.Man )
      I_Contact( #CIn.Manager.Control_ON )
      Contact( #Sts.OP_Manip_CanMoveFreely )
   END_RUNG wire#w1
   RUNG wire#powerrail
      Contact( #CIn.Manager.Sollevamento.Work )
      wire#w2
      Coil( #Sts.Sollevamento.Op_Work_Cnd )
   END_RUNG
   RUNG wire#powerrail
      Contact( #AreaInterface.Man )
      I_Contact( #CIn.Manager.Control_ON )
      Contact( #Sts.OP_Manip_CanMoveFreely )
   END_RUNG wire#w2
   // the same network as SCL:
   #Sts.Sollevamento.OP_Rest_Cnd := #CIn.Manager.Sollevamento.Rest OR (#AreaInterface.Man AND NOT #CIn.Manager.Control_ON AND #Sts.OP_Manip_CanMoveFreely);
   #Sts.Sollevamento.Op_Work_Cnd := #CIn.Manager.Sollevamento.Work OR (#AreaInterface.Man AND NOT #CIn.Manager.Control_ON AND #Sts.OP_Manip_CanMoveFreely);
END_REGION

REGION Network 25: [Magneti] - Condizioni movimento Operazione a Lavoro / Riposo
   RUNG wire#powerrail
      Contact( #CIn.Manager.Magneti.Rest )
      wire#w1
      Coil( #Sts.Magneti.OP_Rest_Cnd )
   END_RUNG
   RUNG wire#powerrail
      Contact( #AreaInterface.Man )
      I_Contact( #CIn.Manager.Control_ON )
      Contact( #Sts.OP_Manip_CanMoveFreely )
   END_RUNG wire#w1
   RUNG wire#powerrail
      Contact( #CIn.Manager.Magneti.Work )
      wire#w2
      Coil( #Sts.Magneti.Op_Work_Cnd )
   END_RUNG
   RUNG wire#powerrail
      Contact( #AreaInterface.Man )
      I_Contact( #CIn.Manager.Control_ON )
      Contact( #Sts.OP_Manip_CanMoveFreely )
   END_RUNG wire#w2
   // the same network as SCL:
   #Sts.Magneti.OP_Rest_Cnd := #CIn.Manager.Magneti.Rest OR (#AreaInterface.Man AND NOT #CIn.Manager.Control_ON AND #Sts.OP_Manip_CanMoveFreely);
   #Sts.Magneti.Op_Work_Cnd := #CIn.Manager.Magneti.Work OR (#AreaInterface.Man AND NOT #CIn.Manager.Control_ON AND #Sts.OP_Manip_CanMoveFreely);
END_REGION

REGION Network 26: <+>
END_REGION

REGION Network 27 (SCL): Manipolatore - CIn Abilitazioni Stop Manager
   // Manipolatore testa
   #Magnete_Testa.Cin.Manager.EnableStopDoorOpeningReq := #Sollevatore_Testa.Cin.Manager.EnableStopDoorOpeningReq
   := #Ax_Testa.CIn.Manager.EnableStopDoorOpeningReq := #CIn.Manager.EnableStopDoorOpeningReq;

   #Magnete_Testa.Cin.Manager.EnableStopInPhase := #Sollevatore_Testa.Cin.Manager.EnableStopInPhase
   := #Ax_Testa.CIn.Manager.EnableStopInPhase := #CIn.Manager.EnableStopInPhase;

   #Magnete_Testa.Cin.Manager.EnableStopProgrammed := #Sollevatore_Testa.Cin.Manager.EnableStopProgrammed
   := #Ax_Testa.CIn.Manager.EnableStopProgrammed := #CIn.Manager.EnableStopProgrammed;

   // Manipolatore coda
   #Magnete_Coda.Cin.Manager.EnableStopDoorOpeningReq := #Sollevatore_Coda.Cin.Manager.EnableStopDoorOpeningReq
   := #Ax_Coda.CIn.Manager.EnableStopDoorOpeningReq := #CIn.Manager.EnableStopDoorOpeningReq;

   #Magnete_Coda.Cin.Manager.EnableStopInPhase := #Sollevatore_Coda.Cin.Manager.EnableStopInPhase
   := #Ax_Coda.CIn.Manager.EnableStopInPhase := #CIn.Manager.EnableStopInPhase;

   #Magnete_Coda.Cin.Manager.EnableStopProgrammed := #Sollevatore_Coda.Cin.Manager.EnableStopProgrammed
   := #Ax_Coda.CIn.Manager.EnableStopProgrammed := #CIn.Manager.EnableStopProgrammed;
END_REGION

REGION Network 28: <+>
END_REGION

REGION Network 29: <<< MANIP TESTA >>>
END_REGION

REGION Network 30: [Ax] HMI preset position
   RUNG wire#powerrail
      Contact( #HMI.Ax_Testa.PbPreset )
      Coil( #Ax_Testa.HMI.B_Preset )
   END_RUNG
   RUNG wire#powerrail
      Move(in := #HMI.Ax_Testa.PresetValue, out1 => #Ax_Testa.HMI.PresetPosition)
   END_RUNG
   // the same network as SCL:
   #Ax_Testa.HMI.B_Preset := #HMI.Ax_Testa.PbPreset;
   #Ax_Testa.HMI.PresetPosition := #HMI.Ax_Testa.PresetValue;
END_REGION

REGION Network 31: [Ax] Axis Manager
   RUNG wire#powerrail
      #Ax_Testa(AreaInterface := #AreaInterface, ZSI := #ZSI, DSI := #DSI_Testa_Feed, Drive := #Drive_Testa, DataIn :=, CIn :=, Config := #Config.Testa.Ax, HW_ID_TEL111 := #HWID_AxTesta_TEL111, Par := #Par.Ax, Pers_Data := #Pers_Data, Warning := #Warning.Testa.Ax, Alarm := #Alarm.Testa.Ax, MachineInterface =>, DataOut =>, COut => #COut.Testa.Ax)
   END_RUNG
   // the same network as SCL:
   #Ax_Testa(AreaInterface := #AreaInterface,   // "Positioning_EPOS_Machine_FB_NEW"
             ZSI := #ZSI,
             DSI := #DSI_Testa_Feed,
             Drive := #Drive_Testa,
             Config := #Config.Testa.Ax,
             HW_ID_TEL111 := #HWID_AxTesta_TEL111,
             Par := #Par.Ax,
             Pers_Data := #Pers_Data,
             Warning := #Warning.Testa.Ax,
             Alarm := #Alarm.Testa.Ax,
             COut => #COut.Testa.Ax);
END_REGION

REGION Network 32: [Sollevatore] - Valve Manager
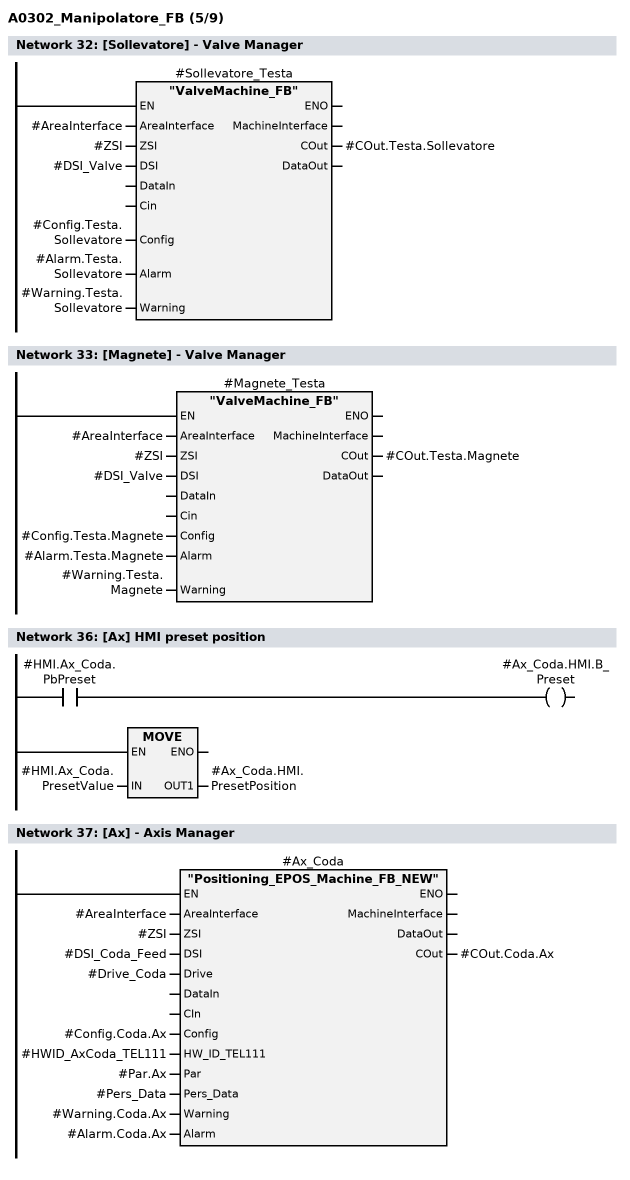
   RUNG wire#powerrail
      #Sollevatore_Testa(AreaInterface := #AreaInterface, ZSI := #ZSI, DSI := #DSI_Valve, DataIn :=, Cin :=, Config := #Config.Testa.Sollevatore, Alarm := #Alarm.Testa.Sollevatore, Warning := #Warning.Testa.Sollevatore, MachineInterface =>, COut => #COut.Testa.Sollevatore, DataOut =>)
   END_RUNG
   // the same network as SCL:
   #Sollevatore_Testa(AreaInterface := #AreaInterface,   // "ValveMachine_FB"
                      ZSI := #ZSI,
                      DSI := #DSI_Valve,
                      Config := #Config.Testa.Sollevatore,
                      Alarm := #Alarm.Testa.Sollevatore,
                      Warning := #Warning.Testa.Sollevatore,
                      COut => #COut.Testa.Sollevatore);
END_REGION

REGION Network 33: [Magnete] - Valve Manager
   RUNG wire#powerrail
      #Magnete_Testa(AreaInterface := #AreaInterface, ZSI := #ZSI, DSI := #DSI_Valve, DataIn :=, Cin :=, Config := #Config.Testa.Magnete, Alarm := #Alarm.Testa.Magnete, Warning := #Warning.Testa.Magnete, MachineInterface =>, COut => #COut.Testa.Magnete, DataOut =>)
   END_RUNG
   // the same network as SCL:
   #Magnete_Testa(AreaInterface := #AreaInterface,   // "ValveMachine_FB"
                  ZSI := #ZSI,
                  DSI := #DSI_Valve,
                  Config := #Config.Testa.Magnete,
                  Alarm := #Alarm.Testa.Magnete,
                  Warning := #Warning.Testa.Magnete,
                  COut => #COut.Testa.Magnete);
END_REGION

REGION Network 35: <<< MANIP CODA>>>
END_REGION

REGION Network 36: [Ax] HMI preset position
   RUNG wire#powerrail
      Contact( #HMI.Ax_Coda.PbPreset )
      Coil( #Ax_Coda.HMI.B_Preset )
   END_RUNG
   RUNG wire#powerrail
      Move(in := #HMI.Ax_Coda.PresetValue, out1 => #Ax_Coda.HMI.PresetPosition)
   END_RUNG
   // the same network as SCL:
   #Ax_Coda.HMI.B_Preset := #HMI.Ax_Coda.PbPreset;
   #Ax_Coda.HMI.PresetPosition := #HMI.Ax_Coda.PresetValue;
END_REGION

REGION Network 37: [Ax] - Axis Manager
   RUNG wire#powerrail
      #Ax_Coda(AreaInterface := #AreaInterface, ZSI := #ZSI, DSI := #DSI_Coda_Feed, Drive := #Drive_Coda, DataIn :=, CIn :=, Config := #Config.Coda.Ax, HW_ID_TEL111 := #HWID_AxCoda_TEL111, Par := #Par.Ax, Pers_Data := #Pers_Data, Warning := #Warning.Coda.Ax, Alarm := #Alarm.Coda.Ax, MachineInterface =>, DataOut =>, COut => #COut.Coda.Ax)
   END_RUNG
   // the same network as SCL:
   #Ax_Coda(AreaInterface := #AreaInterface,   // "Positioning_EPOS_Machine_FB_NEW"
            ZSI := #ZSI,
            DSI := #DSI_Coda_Feed,
            Drive := #Drive_Coda,
            Config := #Config.Coda.Ax,
            HW_ID_TEL111 := #HWID_AxCoda_TEL111,
            Par := #Par.Ax,
            Pers_Data := #Pers_Data,
            Warning := #Warning.Coda.Ax,
            Alarm := #Alarm.Coda.Ax,
            COut => #COut.Coda.Ax);
END_REGION

REGION Network 38: [Sollevatore] - Valve Manager
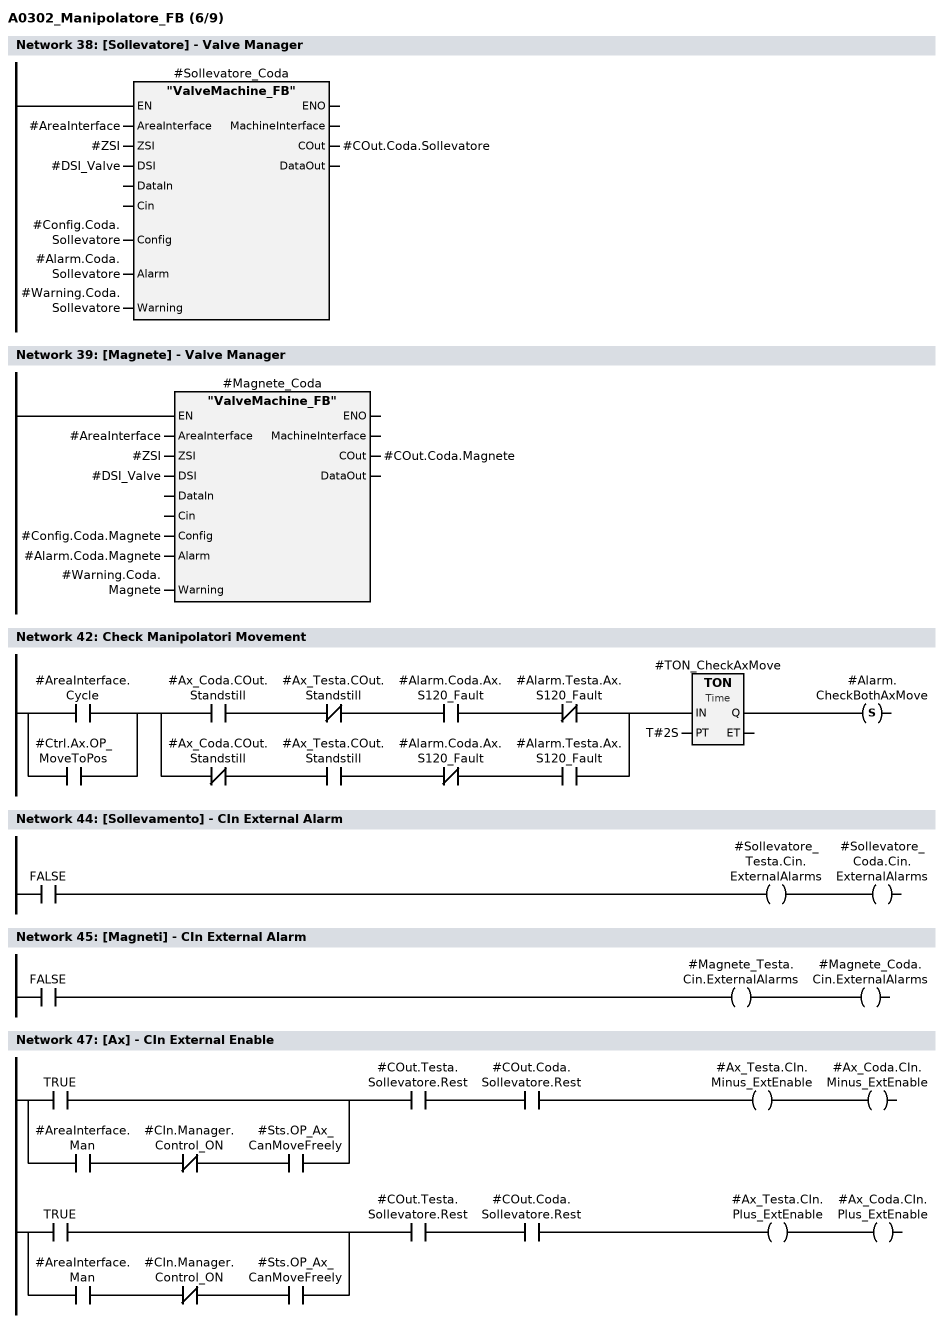
   RUNG wire#powerrail
      #Sollevatore_Coda(AreaInterface := #AreaInterface, ZSI := #ZSI, DSI := #DSI_Valve, DataIn :=, Cin :=, Config := #Config.Coda.Sollevatore, Alarm := #Alarm.Coda.Sollevatore, Warning := #Warning.Coda.Sollevatore, MachineInterface =>, COut => #COut.Coda.Sollevatore, DataOut =>)
   END_RUNG
   // the same network as SCL:
   #Sollevatore_Coda(AreaInterface := #AreaInterface,   // "ValveMachine_FB"
                     ZSI := #ZSI,
                     DSI := #DSI_Valve,
                     Config := #Config.Coda.Sollevatore,
                     Alarm := #Alarm.Coda.Sollevatore,
                     Warning := #Warning.Coda.Sollevatore,
                     COut => #COut.Coda.Sollevatore);
END_REGION

REGION Network 39: [Magnete] - Valve Manager
   RUNG wire#powerrail
      #Magnete_Coda(AreaInterface := #AreaInterface, ZSI := #ZSI, DSI := #DSI_Valve, DataIn :=, Cin :=, Config := #Config.Coda.Magnete, Alarm := #Alarm.Coda.Magnete, Warning := #Warning.Coda.Magnete, MachineInterface =>, COut => #COut.Coda.Magnete, DataOut =>)
   END_RUNG
   // the same network as SCL:
   #Magnete_Coda(AreaInterface := #AreaInterface,   // "ValveMachine_FB"
                 ZSI := #ZSI,
                 DSI := #DSI_Valve,
                 Config := #Config.Coda.Magnete,
                 Alarm := #Alarm.Coda.Magnete,
                 Warning := #Warning.Coda.Magnete,
                 COut => #COut.Coda.Magnete);
END_REGION

REGION Network 41 (SCL): Sincronizzazione tra asse testa e asse coda
   #CheckAxisSynch(Ax1_Pos:=#Ax_Testa.Sts.ActualPosition,
                   Ax2_Pos:=#Ax_Coda.Sts.ActualPosition,
                   TargetPos:=#Ax_Testa.Ctrl.Pos,
                   MaxDistance:=#MaxDistance,
                   MinDistance:=#MinDistance,
                   Ax1_SynchOk=> #Sts.Testa_PermessoDaSynchOk,
                   Ax2_SynchOk=> #Sts.Coda_PermessoDaSynchOk);
END_REGION

REGION Network 42: Check Manipolatori Movement
   RUNG wire#powerrail
      Contact( #AreaInterface.Cycle )
      wire#w1
      Contact( #Ax_Coda.COut.Standstill )
      I_Contact( #Ax_Testa.COut.Standstill )
      Contact( #Alarm.Coda.Ax.S120_Fault )
      I_Contact( #Alarm.Testa.Ax.S120_Fault )
      wire#w2
      { S7_Templates := "time_type := Time" } #TON_CheckAxMove.TON(pt := T#2S, et =>)
      S_Coil( #Alarm.CheckBothAxMove )
   END_RUNG
   RUNG wire#powerrail
      Contact( #Ctrl.Ax.OP_MoveToPos )
   END_RUNG wire#w1
   RUNG wire#w1
      I_Contact( #Ax_Coda.COut.Standstill )
      Contact( #Ax_Testa.COut.Standstill )
      I_Contact( #Alarm.Coda.Ax.S120_Fault )
      Contact( #Alarm.Testa.Ax.S120_Fault )
   END_RUNG wire#w2
   // the same network as SCL:
   #TON_CheckAxMove.TON(IN := (#AreaInterface.Cycle OR #Ctrl.Ax.OP_MoveToPos) AND ((#Ax_Coda.COut.Standstill AND NOT #Ax_Testa.COut.Standstill AND #Alarm.Coda.Ax.S120_Fault AND NOT #Alarm.Testa.Ax.S120_Fault) OR (NOT #Ax_Coda.COut.Standstill AND #Ax_Testa.COut.Standstill AND NOT #Alarm.Coda.Ax.S120_Fault AND #Alarm.Testa.Ax.S120_Fault)),
                        PT := T#2S);
   IF #TON_CheckAxMove.Q THEN #Alarm.CheckBothAxMove := TRUE; END_IF;
END_REGION

REGION Network 44: [Sollevamento] - CIn External Alarm
   RUNG wire#powerrail
      Contact( FALSE )
      Coil( #Sollevatore_Testa.Cin.ExternalAlarms )
      Coil( #Sollevatore_Coda.Cin.ExternalAlarms )
   END_RUNG
   // the same network as SCL:
   #Sollevatore_Testa.Cin.ExternalAlarms := FALSE;
   #Sollevatore_Coda.Cin.ExternalAlarms := FALSE;
END_REGION

REGION Network 45: [Magneti] - CIn External Alarm
   RUNG wire#powerrail
      Contact( FALSE )
      Coil( #Magnete_Testa.Cin.ExternalAlarms )
      Coil( #Magnete_Coda.Cin.ExternalAlarms )
   END_RUNG
   // the same network as SCL:
   #Magnete_Testa.Cin.ExternalAlarms := FALSE;
   #Magnete_Coda.Cin.ExternalAlarms := FALSE;
END_REGION

REGION Network 46: <+>
END_REGION

REGION Network 47: [Ax] - CIn External Enable
   RUNG wire#powerrail
      Contact( TRUE )
      wire#w1
      Contact( #COut.Testa.Sollevatore.Rest )
      Contact( #COut.Coda.Sollevatore.Rest )
      Coil( #Ax_Testa.CIn.Minus_ExtEnable )
      Coil( #Ax_Coda.CIn.Minus_ExtEnable )
   END_RUNG
   RUNG wire#powerrail
      Contact( #AreaInterface.Man )
      I_Contact( #CIn.Manager.Control_ON )
      Contact( #Sts.OP_Ax_CanMoveFreely )
   END_RUNG wire#w1
   RUNG wire#powerrail
      Contact( TRUE )
      wire#w2
      Contact( #COut.Testa.Sollevatore.Rest )
      Contact( #COut.Coda.Sollevatore.Rest )
      Coil( #Ax_Testa.CIn.Plus_ExtEnable )
      Coil( #Ax_Coda.CIn.Plus_ExtEnable )
   END_RUNG
   RUNG wire#powerrail
      Contact( #AreaInterface.Man )
      I_Contact( #CIn.Manager.Control_ON )
      Contact( #Sts.OP_Ax_CanMoveFreely )
   END_RUNG wire#w2
   // the same network as SCL:
   #Ax_Testa.CIn.Minus_ExtEnable := (TRUE OR (#AreaInterface.Man AND NOT #CIn.Manager.Control_ON AND #Sts.OP_Ax_CanMoveFreely)) AND #COut.Testa.Sollevatore.Rest AND #COut.Coda.Sollevatore.Rest;
   #Ax_Coda.CIn.Minus_ExtEnable := #Ax_Testa.CIn.Minus_ExtEnable;
   #Ax_Testa.CIn.Plus_ExtEnable := (TRUE OR (#AreaInterface.Man AND NOT #CIn.Manager.Control_ON AND #Sts.OP_Ax_CanMoveFreely)) AND #COut.Testa.Sollevatore.Rest AND #COut.Coda.Sollevatore.Rest;
   #Ax_Coda.CIn.Plus_ExtEnable := #Ax_Testa.CIn.Plus_ExtEnable;
END_REGION

REGION Network 48: [Sollevamento] - CIn External Enable
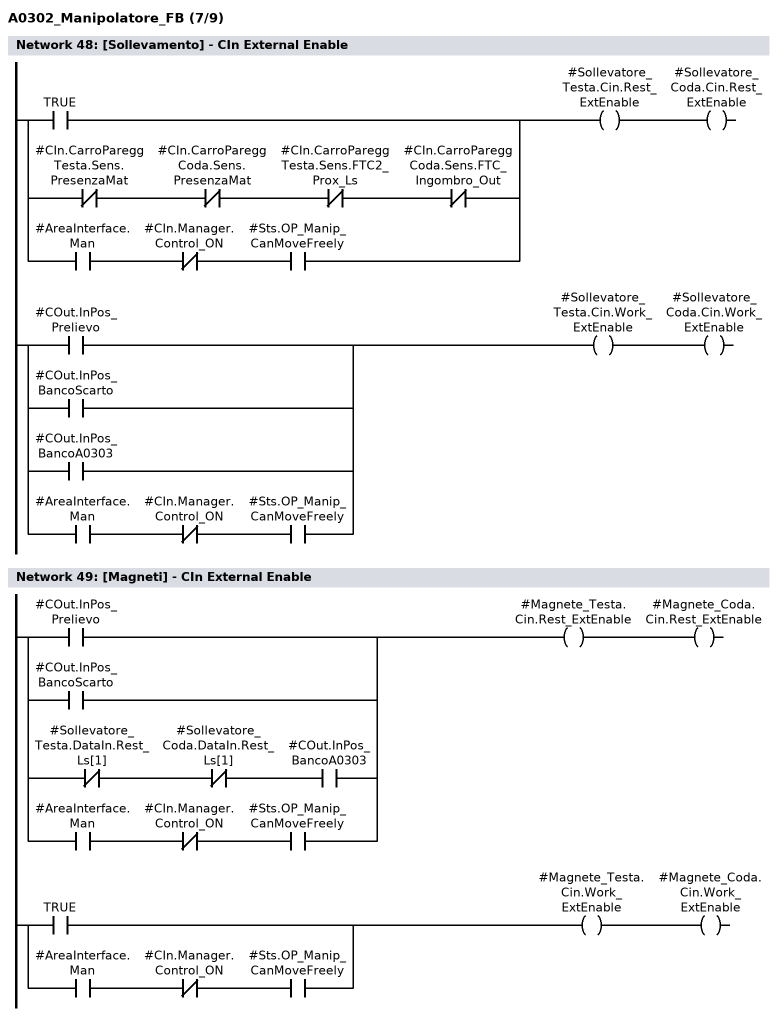
   RUNG wire#powerrail
      Contact( TRUE )
      wire#w1
      Coil( #Sollevatore_Testa.Cin.Rest_ExtEnable )
      Coil( #Sollevatore_Coda.Cin.Rest_ExtEnable )
   END_RUNG
   RUNG wire#powerrail
      I_Contact( #CIn.CarroPareggTesta.Sens.PresenzaMat )
      I_Contact( #CIn.CarroPareggCoda.Sens.PresenzaMat )
      I_Contact( #CIn.CarroPareggTesta.Sens.FTC2_Prox_Ls )
      I_Contact( #CIn.CarroPareggCoda.Sens.FTC_Ingombro_Out )
   END_RUNG wire#w1
   RUNG wire#powerrail
      Contact( #AreaInterface.Man )
      I_Contact( #CIn.Manager.Control_ON )
      Contact( #Sts.OP_Manip_CanMoveFreely )
   END_RUNG wire#w1
   RUNG wire#powerrail
      Contact( #COut.InPos_Prelievo )
      wire#w2
      Coil( #Sollevatore_Testa.Cin.Work_ExtEnable )
      Coil( #Sollevatore_Coda.Cin.Work_ExtEnable )
   END_RUNG
   RUNG wire#powerrail
      Contact( #COut.InPos_BancoScarto )
   END_RUNG wire#w2
   RUNG wire#powerrail
      Contact( #COut.InPos_BancoA0303 )
   END_RUNG wire#w2
   RUNG wire#powerrail
      Contact( #AreaInterface.Man )
      I_Contact( #CIn.Manager.Control_ON )
      Contact( #Sts.OP_Manip_CanMoveFreely )
   END_RUNG wire#w2
   // the same network as SCL:
   #Sollevatore_Testa.Cin.Rest_ExtEnable := TRUE OR (NOT #CIn.CarroPareggTesta.Sens.PresenzaMat AND NOT #CIn.CarroPareggCoda.Sens.PresenzaMat AND NOT #CIn.CarroPareggTesta.Sens.FTC2_Prox_Ls AND NOT #CIn.CarroPareggCoda.Sens.FTC_Ingombro_Out) OR (#AreaInterface.Man AND NOT #CIn.Manager.Control_ON AND #Sts.OP_Manip_CanMoveFreely);
   #Sollevatore_Coda.Cin.Rest_ExtEnable := #Sollevatore_Testa.Cin.Rest_ExtEnable;
   #Sollevatore_Testa.Cin.Work_ExtEnable := #COut.InPos_Prelievo OR #COut.InPos_BancoScarto OR #COut.InPos_BancoA0303 OR (#AreaInterface.Man AND NOT #CIn.Manager.Control_ON AND #Sts.OP_Manip_CanMoveFreely);
   #Sollevatore_Coda.Cin.Work_ExtEnable := #Sollevatore_Testa.Cin.Work_ExtEnable;
END_REGION

REGION Network 49: [Magneti] - CIn External Enable
   RUNG wire#powerrail
      Contact( #COut.InPos_Prelievo )
      wire#w1
      Coil( #Magnete_Testa.Cin.Rest_ExtEnable )
      Coil( #Magnete_Coda.Cin.Rest_ExtEnable )
   END_RUNG
   RUNG wire#powerrail
      Contact( #COut.InPos_BancoScarto )
   END_RUNG wire#w1
   RUNG wire#powerrail
      I_Contact( #Sollevatore_Testa.DataIn.Rest_Ls[1] )
      I_Contact( #Sollevatore_Coda.DataIn.Rest_Ls[1] )
      Contact( #COut.InPos_BancoA0303 )
   END_RUNG wire#w1
   RUNG wire#powerrail
      Contact( #AreaInterface.Man )
      I_Contact( #CIn.Manager.Control_ON )
      Contact( #Sts.OP_Manip_CanMoveFreely )
   END_RUNG wire#w1
   RUNG wire#powerrail
      Contact( TRUE )
      wire#w2
      Coil( #Magnete_Testa.Cin.Work_ExtEnable )
      Coil( #Magnete_Coda.Cin.Work_ExtEnable )
   END_RUNG
   RUNG wire#powerrail
      Contact( #AreaInterface.Man )
      I_Contact( #CIn.Manager.Control_ON )
      Contact( #Sts.OP_Manip_CanMoveFreely )
   END_RUNG wire#w2
   // the same network as SCL:
   #Magnete_Testa.Cin.Rest_ExtEnable := #COut.InPos_Prelievo OR #COut.InPos_BancoScarto OR (NOT #Sollevatore_Testa.DataIn.Rest_Ls[1] AND NOT #Sollevatore_Coda.DataIn.Rest_Ls[1] AND #COut.InPos_BancoA0303) OR (#AreaInterface.Man AND NOT #CIn.Manager.Control_ON AND #Sts.OP_Manip_CanMoveFreely);
   #Magnete_Coda.Cin.Rest_ExtEnable := #Magnete_Testa.Cin.Rest_ExtEnable;
   #Magnete_Testa.Cin.Work_ExtEnable := TRUE OR (#AreaInterface.Man AND NOT #CIn.Manager.Control_ON AND #Sts.OP_Manip_CanMoveFreely);
   #Magnete_Coda.Cin.Work_ExtEnable := #Magnete_Testa.Cin.Work_ExtEnable;
END_REGION

REGION Network 51: [Sollevamento] - Warning mancanza condizioni esecuzione Operazione RIPOSO / LAVORO
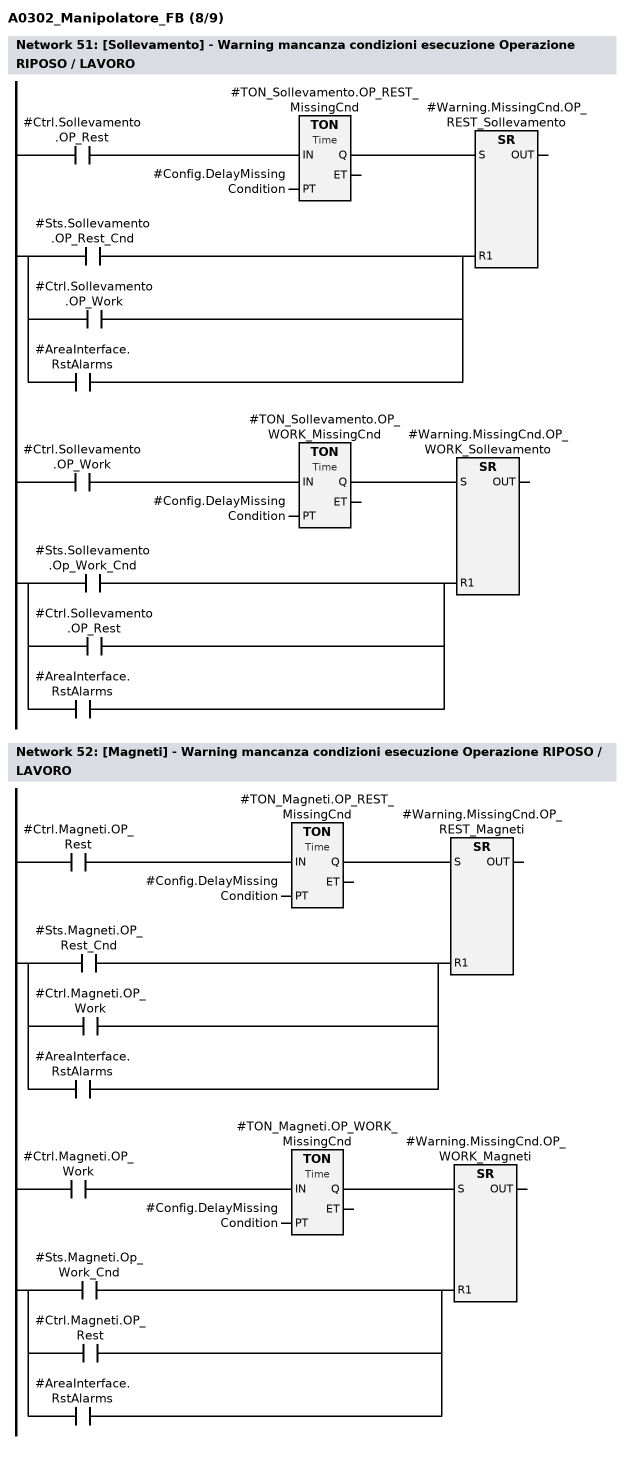
   RUNG wire#powerrail
      Contact( #Ctrl.Sollevamento.OP_Rest )
      { S7_Templates := "time_type := Time" } #TON_Sollevamento.OP_REST_MissingCnd.TON(pt := #Config.DelayMissingCondition, et =>)
      S_SR(operand := #Warning.MissingCnd.OP_REST_Sollevamento, r1 := wire#w1)
   END_RUNG
   RUNG wire#powerrail
      Contact( #Sts.Sollevamento.OP_Rest_Cnd )
   END_RUNG wire#w1
   RUNG wire#powerrail
      Contact( #Ctrl.Sollevamento.OP_Work )
   END_RUNG wire#w1
   RUNG wire#powerrail
      Contact( #AreaInterface.RstAlarms )
   END_RUNG wire#w1
   RUNG wire#powerrail
      Contact( #Ctrl.Sollevamento.OP_Work )
      { S7_Templates := "time_type := Time" } #TON_Sollevamento.OP_WORK_MissingCnd.TON(pt := #Config.DelayMissingCondition, et =>)
      S_SR(operand := #Warning.MissingCnd.OP_WORK_Sollevamento, r1 := wire#w2)
   END_RUNG
   RUNG wire#powerrail
      Contact( #Sts.Sollevamento.Op_Work_Cnd )
   END_RUNG wire#w2
   RUNG wire#powerrail
      Contact( #Ctrl.Sollevamento.OP_Rest )
   END_RUNG wire#w2
   RUNG wire#powerrail
      Contact( #AreaInterface.RstAlarms )
   END_RUNG wire#w2
   // the same network as SCL:
   #TON_Sollevamento.OP_REST_MissingCnd.TON(IN := #Ctrl.Sollevamento.OP_Rest,
                           PT := #Config.DelayMissingCondition);
   IF #TON_Sollevamento.OP_REST_MissingCnd.Q THEN
       #Warning.MissingCnd.OP_REST_Sollevamento := TRUE;   // SR flip-flop
   END_IF;
   IF #Sts.Sollevamento.OP_Rest_Cnd OR #Ctrl.Sollevamento.OP_Work OR #AreaInterface.RstAlarms THEN
       #Warning.MissingCnd.OP_REST_Sollevamento := FALSE;
   END_IF;
   #TON_Sollevamento.OP_WORK_MissingCnd.TON(IN := #Ctrl.Sollevamento.OP_Work,
                           PT := #Config.DelayMissingCondition);
   IF #TON_Sollevamento.OP_WORK_MissingCnd.Q THEN
       #Warning.MissingCnd.OP_WORK_Sollevamento := TRUE;   // SR flip-flop
   END_IF;
   IF #Sts.Sollevamento.Op_Work_Cnd OR #Ctrl.Sollevamento.OP_Rest OR #AreaInterface.RstAlarms THEN
       #Warning.MissingCnd.OP_WORK_Sollevamento := FALSE;
   END_IF;
END_REGION

REGION Network 52: [Magneti] - Warning mancanza condizioni esecuzione Operazione RIPOSO / LAVORO
   RUNG wire#powerrail
      Contact( #Ctrl.Magneti.OP_Rest )
      { S7_Templates := "time_type := Time" } #TON_Magneti.OP_REST_MissingCnd.TON(pt := #Config.DelayMissingCondition, et =>)
      S_SR(operand := #Warning.MissingCnd.OP_REST_Magneti, r1 := wire#w1)
   END_RUNG
   RUNG wire#powerrail
      Contact( #Sts.Magneti.OP_Rest_Cnd )
   END_RUNG wire#w1
   RUNG wire#powerrail
      Contact( #Ctrl.Magneti.OP_Work )
   END_RUNG wire#w1
   RUNG wire#powerrail
      Contact( #AreaInterface.RstAlarms )
   END_RUNG wire#w1
   RUNG wire#powerrail
      Contact( #Ctrl.Magneti.OP_Work )
      { S7_Templates := "time_type := Time" } #TON_Magneti.OP_WORK_MissingCnd.TON(pt := #Config.DelayMissingCondition, et =>)
      S_SR(operand := #Warning.MissingCnd.OP_WORK_Magneti, r1 := wire#w2)
   END_RUNG
   RUNG wire#powerrail
      Contact( #Sts.Magneti.Op_Work_Cnd )
   END_RUNG wire#w2
   RUNG wire#powerrail
      Contact( #Ctrl.Magneti.OP_Rest )
   END_RUNG wire#w2
   RUNG wire#powerrail
      Contact( #AreaInterface.RstAlarms )
   END_RUNG wire#w2
   // the same network as SCL:
   #TON_Magneti.OP_REST_MissingCnd.TON(IN := #Ctrl.Magneti.OP_Rest, PT := #Config.DelayMissingCondition);
   IF #TON_Magneti.OP_REST_MissingCnd.Q THEN
       #Warning.MissingCnd.OP_REST_Magneti := TRUE;   // SR flip-flop
   END_IF;
   IF #Sts.Magneti.OP_Rest_Cnd OR #Ctrl.Magneti.OP_Work OR #AreaInterface.RstAlarms THEN
       #Warning.MissingCnd.OP_REST_Magneti := FALSE;
   END_IF;
   #TON_Magneti.OP_WORK_MissingCnd.TON(IN := #Ctrl.Magneti.OP_Work, PT := #Config.DelayMissingCondition);
   IF #TON_Magneti.OP_WORK_MissingCnd.Q THEN
       #Warning.MissingCnd.OP_WORK_Magneti := TRUE;   // SR flip-flop
   END_IF;
   IF #Sts.Magneti.Op_Work_Cnd OR #Ctrl.Magneti.OP_Rest OR #AreaInterface.RstAlarms THEN
       #Warning.MissingCnd.OP_WORK_Magneti := FALSE;
   END_IF;
END_REGION

REGION Network 54 (SCL): [Ax] - Cin Manager (Esecuzione sequenza comandi)
   // Operazione LAVORO dell' asse spintore quando i 2 ciclindri sono in riposo e il bloccaggio è a riposo

   // MANIPOLATORE TESTA
   #Ax_Testa.CIn.Manager.Control_ON := #Sollevatore_Testa.Cin.Manager.Control_ON := #Magnete_Testa.Cin.Manager.Control_ON := #CIn.Manager.Control_ON;
   #Ax_Coda.CIn.Manager.Control_ON := #Sollevatore_Coda.Cin.Manager.Control_ON := #Magnete_Coda.Cin.Manager.Control_ON := #CIn.Manager.Control_ON;

   #Ax_Testa.CIn.Manager.Acc := #Ax_Coda.CIn.Manager.Acc := #CIn.Manager.Acc;
   #Ax_Testa.CIn.Manager.Dec := #Ax_Coda.CIn.Manager.Dec := #CIn.Manager.Dec;
   #Ax_Testa.CIn.Manager.Vel := #Ax_Coda.CIn.Manager.Vel := #CIn.Manager.Vel;

   IF #Sts_PosAxis = 2 AND (NOT #Sts.Testa_PermessoDaSynchOk OR NOT #Sts.Coda_PermessoDaSynchOk) THEN
       #Sts_PosAxis := 0;
   END_IF;

   IF NOT #Ctrl.Ax.OP_MoveToPos THEN
       #Sts_PosAxis := 0;
   END_IF;

   IF #Sts_PosAxis = 0 THEN

       #Ax_Testa.CIn.Manager.MoveToPos := #Ax_Coda.CIn.Manager.MoveToPos := FALSE;

       IF #Ctrl.Ax.OP_MoveToPos THEN

           IF ABS(#Ax_Testa.Sts.ActualPosition - #Ax_Coda.Sts.ActualPosition) > 0.5 THEN
               IF #Ax_Testa.Sts.ActualPosition > #Ax_Coda.Sts.ActualPosition THEN
                   #Ax_Coda.CIn.Manager.Pos := #Ax_Testa.Sts.ActualPosition;
                   #Ax_Coda.CIn.Manager.MoveToPos := TRUE;
               ELSE
                   #Ax_Testa.CIn.Manager.Pos := #Ax_Coda.Sts.ActualPosition;
                   #Ax_Testa.CIn.Manager.MoveToPos := TRUE;
               END_IF;
               #Sts_PosAxis += 1;
           ELSE
               #Sts_PosAxis := 2;
           END_IF;
       END_IF;
   END_IF;

   IF #Sts_PosAxis = 1 THEN

       IF NOT #Ax_Testa.CIn.Manager.MoveToPos AND NOT #Ax_Coda.CIn.Manager.MoveToPos THEN
           #Sts_PosAxis := 0;
       END_IF;


           IF ABS(#Ax_Testa.Sts.ActualPosition - #Ax_Coda.Sts.ActualPosition) < 0.1 THEN
               #Ax_Testa.CIn.Manager.MoveToPos := FALSE;
               #Ax_Coda.CIn.Manager.MoveToPos := FALSE;

               #Sts_PosAxis += 1;

           END_IF;
       END_IF;

       IF #Sts_PosAxis = 2 AND NOT #Alarm.CheckBothAxMove THEN
               //
               #Ax_Testa.CIn.Manager.MoveToPos := #Ctrl.Ax.OP_MoveToPos AND #Sts.Op_MoveToPos_Cnd;
               #Ax_Coda.CIn.Manager.MoveToPos := #Ctrl.Ax.OP_MoveToPos AND #Sts.Op_MoveToPos_Cnd;
               #Ax_Testa.CIn.Manager.Pos := #Ax_Coda.CIn.Manager.Pos := #CIn.Manager.Pos;

       END_IF;


       // ##########################
   (*    
   IF #Ctrl.Ax.OP_MoveToPos AND #Sts.Op_MoveToPos_Cnd AND NOT #Ax_Testa.COut.InPosition AND #Sollevatore_Testa.COut.Rest
       AND ( NOT #Alarm.Testa.Ax.S120_Fault AND NOT #Alarm.Coda.Ax.S120_Fault) THEN
       #Ax_Testa.CIn.Manager.MoveToPos := TRUE;

       // Se raggiungo la posizione di setpoint spengo il comando
   ELSIF #Ax_Testa.COut.InPosition AND #Ax_Testa.COut.Standstill OR ( #Alarm.Testa.Ax.S120_Fault OR #Alarm.Coda.Ax.S120_Fault) THEN
       #Ax_Testa.CIn.Manager.MoveToPos := FALSE;
       #Ax_Testa.DSI.PowerEnable := FALSE;
   END_IF;

   // MANIPOLATORE CODA
   #Ax_Coda.CIn.Manager.Control_ON := #Ax_Coda.DSI.PowerEnable
   := #Sollevatore_Coda.Cin.Manager.Control_ON := #Magnete_Coda.Cin.Manager.Control_ON := #Ctrl.Ax.OP_MoveToPos;

   IF #Ctrl.Ax.OP_MoveToPos AND #Sts.Op_MoveToPos_Cnd AND NOT #Ax_Coda.COut.InPosition AND #Sollevatore_Coda.COut.Rest
       AND ( NOT #Alarm.Testa.Ax.S120_Fault AND NOT #Alarm.Coda.Ax.S120_Fault) THEN
           #Ax_Coda.CIn.Manager.MoveToPos := TRUE;

           // Se raggiungo la posizione di setpoint spengo il comando
       ELSIF #Ax_Coda.COut.InPosition AND #Ax_Coda.COut.Standstill OR ( #Alarm.Testa.Ax.S120_Fault OR #Alarm.Coda.Ax.S120_Fault) THEN
           #Ax_Coda.CIn.Manager.MoveToPos := FALSE;
           #Ax_Coda.DSI.PowerEnable := FALSE;
       END_IF;
       *)
END_REGION

REGION Network 55 (SCL): [Sollevamento] - Cin Manager (Esecuzione sequenza comandi)
   // Comando CIn Manager ControlON di tutte le utenze
   // MANIPOLATORE TESTA & CODA
   #Sollevatore_Testa.Cin.Manager.Control_ON := #CIn.Manager.Control_ON;
   #Sollevatore_Coda.Cin.Manager.Control_ON := #CIn.Manager.Control_ON;
   //
   #Sollevatore_Testa.Cin.Manager.Rest := FALSE;
   #Sollevatore_Testa.Cin.Manager.Work := FALSE;
   #Sollevatore_Coda.Cin.Manager.Rest := FALSE;
   #Sollevatore_Coda.Cin.Manager.Work := FALSE;

   // Gestione dei comandi relativi a Sollevamento in sequenza quando ho un OP cnd

   IF (#Ctrl.Sollevamento.OP_Rest AND #Sts.Sollevamento.OP_Rest_Cnd) THEN

       #Sollevatore_Testa.Cin.Manager.Rest := TRUE;
       #Sollevatore_Coda.Cin.Manager.Rest := TRUE;

           // Vado a lavoro solo se sono in posizione    
   ELSIF  (#Ctrl.Sollevamento.OP_Work AND #Sts.Sollevamento.Op_Work_Cnd) AND (#COut.InPos_Prelievo OR #COut.InPos_BancoScarto OR #COut.InPos_BancoA0303) THEN

       #Sollevatore_Testa.Cin.Manager.Work := TRUE;
       #Sollevatore_Coda.Cin.Manager.Work := TRUE;

   END_IF;
END_REGION

REGION Network 56 (SCL): [Magneti] - Cin Manager (Esecuzione sequenza comandi)


   // Comando CIn Manager ControlON di tutte le utenze
   // MAGNETI TESTA & CODA
   #Magnete_Testa.Cin.Manager.Control_ON := (#Ctrl.Magneti.OP_Rest OR #Ctrl.Magneti.OP_Work) OR (#Ctrl.Sollevamento.OP_Rest OR #Ctrl.Sollevamento.OP_Work);
   #Magnete_Coda.Cin.Manager.Control_ON := (#Ctrl.Magneti.OP_Rest OR #Ctrl.Magneti.OP_Work) OR (#Ctrl.Sollevamento.OP_Rest OR #Ctrl.Sollevamento.OP_Work);
   //
   // Gestione dei comandi relativi ai Magneti in sequenza quando ho un OP cnd
   IF (#Ctrl.Magneti.OP_Rest AND #Sts.Magneti.OP_Rest_Cnd) AND #Sollevatore_Testa.COut.Work AND #Sollevatore_Coda.COut.Work THEN

       #Magnete_Testa.Cin.Manager.Work := FALSE;
       #Magnete_Coda.Cin.Manager.Work := FALSE;
       #Magnete_Testa.Cin.Manager.Rest := TRUE;
       #Magnete_Coda.Cin.Manager.Rest := TRUE;

   ELSIF (#Ctrl.Magneti.OP_Rest AND #Sts.Magneti.OP_Rest_Cnd) AND #COut.InPos_BancoScarto THEN

       #Magnete_Testa.Cin.Manager.Work := FALSE;
       #Magnete_Coda.Cin.Manager.Work := FALSE;
       #Magnete_Testa.Cin.Manager.Rest := TRUE;
       #Magnete_Coda.Cin.Manager.Rest := TRUE;

           // Vado a lavoro solo se sono in posizione e il sollevatore è a lavoro    
   ELSIF  (#Ctrl.Magneti.OP_Work AND #Sts.Magneti.Op_Work_Cnd) THEN

       #Magnete_Testa.Cin.Manager.Rest := FALSE;
       #Magnete_Coda.Cin.Manager.Rest := FALSE;
       #Magnete_Testa.Cin.Manager.Work := TRUE;
       #Magnete_Coda.Cin.Manager.Work := TRUE;

   END_IF;
END_REGION

REGION Network 58: <<< MACHINE STATUS >>>
END_REGION

REGION Network 59: Collect machine to zone interface (internal machines OR)
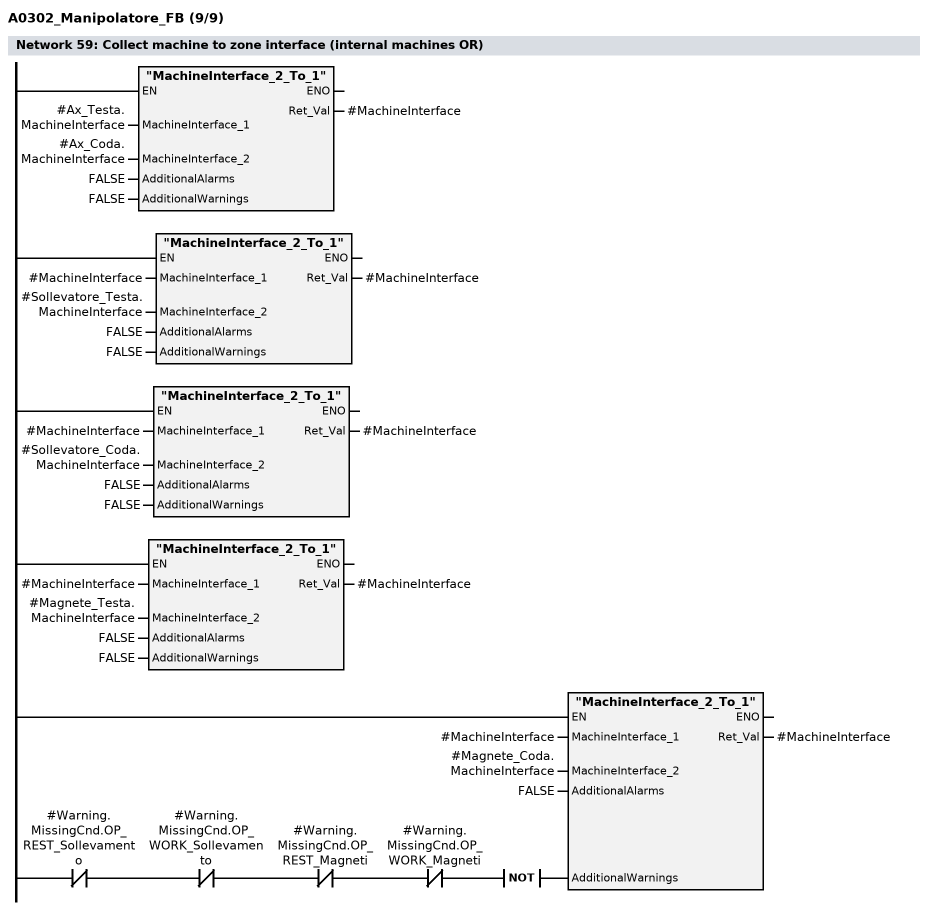
   RUNG wire#powerrail
      "MachineInterface_2_To_1"(MachineInterface_1 := #Ax_Testa.MachineInterface, MachineInterface_2 := #Ax_Coda.MachineInterface, AdditionalAlarms := FALSE, AdditionalWarnings := FALSE, Ret_Val => #MachineInterface)
   END_RUNG
   RUNG wire#powerrail
      "MachineInterface_2_To_1"(MachineInterface_1 := #MachineInterface, MachineInterface_2 := #Sollevatore_Testa.MachineInterface, AdditionalAlarms := FALSE, AdditionalWarnings := FALSE, Ret_Val => #MachineInterface)
   END_RUNG
   RUNG wire#powerrail
      "MachineInterface_2_To_1"(MachineInterface_1 := #MachineInterface, MachineInterface_2 := #Sollevatore_Coda.MachineInterface, AdditionalAlarms := FALSE, AdditionalWarnings := FALSE, Ret_Val => #MachineInterface)
   END_RUNG
   RUNG wire#powerrail
      "MachineInterface_2_To_1"(MachineInterface_1 := #MachineInterface, MachineInterface_2 := #Magnete_Testa.MachineInterface, AdditionalAlarms := FALSE, AdditionalWarnings := FALSE, Ret_Val => #MachineInterface)
   END_RUNG
   RUNG wire#powerrail
      "MachineInterface_2_To_1"(AdditionalWarnings := wire#w1, MachineInterface_1 := #MachineInterface, MachineInterface_2 := #Magnete_Coda.MachineInterface, AdditionalAlarms := FALSE, Ret_Val => #MachineInterface)
   END_RUNG
   RUNG wire#powerrail
      I_Contact( #Warning.MissingCnd.OP_REST_Sollevamento )
      I_Contact( #Warning.MissingCnd.OP_WORK_Sollevamento )
      I_Contact( #Warning.MissingCnd.OP_REST_Magneti )
      I_Contact( #Warning.MissingCnd.OP_WORK_Magneti )
      Not()
   END_RUNG wire#w1
   // the same network as SCL:
   #MachineInterface := "MachineInterface_2_To_1"(MachineInterface_1 := #Ax_Testa.MachineInterface,
                           MachineInterface_2 := #Ax_Coda.MachineInterface,
                           AdditionalAlarms := FALSE,
                           AdditionalWarnings := FALSE);
   #MachineInterface := "MachineInterface_2_To_1"(MachineInterface_1 := #MachineInterface,
                           MachineInterface_2 := #Sollevatore_Testa.MachineInterface,
                           AdditionalAlarms := FALSE,
                           AdditionalWarnings := FALSE);
   #MachineInterface := "MachineInterface_2_To_1"(MachineInterface_1 := #MachineInterface,
                           MachineInterface_2 := #Sollevatore_Coda.MachineInterface,
                           AdditionalAlarms := FALSE,
                           AdditionalWarnings := FALSE);
   #MachineInterface := "MachineInterface_2_To_1"(MachineInterface_1 := #MachineInterface,
                           MachineInterface_2 := #Magnete_Testa.MachineInterface,
                           AdditionalAlarms := FALSE,
                           AdditionalWarnings := FALSE);
   #MachineInterface := "MachineInterface_2_To_1"(MachineInterface_1 := #MachineInterface,
                           MachineInterface_2 := #Magnete_Coda.MachineInterface,
                           AdditionalAlarms := FALSE,
                           AdditionalWarnings := NOT (NOT #Warning.MissingCnd.OP_REST_Sollevamento AND NOT #Warning.MissingCnd.OP_WORK_Sollevamento AND NOT #Warning.MissingCnd.OP_REST_Magneti AND NOT #Warning.MissingCnd.OP_WORK_Magneti));
END_REGION
END_FUNCTION_BLOCK
